// TIA Portal V18 export
ORGANIZATION_BLOCK "Work Cyclic"   // OB30, LAD, CyclicInterrupt
TITLE = Description:
{ S7_Optimized_Access := 'TRUE' }
VERSION : 0.1
// Operations that are supposed to be executed in a precise cycle time, which is temporary set to 45ms. It is important to connect this time with the read/write time of the WebDB (NOAH).
// stored: AutoNumber true, IsIECCheckEnabled false, SetENOAutomatically false
   VAR_INPUT
      Initial_Call : Bool;   // Initial call of this OB
      Event_Count : Int;   // Events discarded
   END_VAR
   VAR_TEMP   // added for the SCL form of the ladder/FBD networks
      _w1 : Bool;
   END_VAR
BEGIN

REGION Network 1: AXIS Z1 Control CMMT V2 To Update
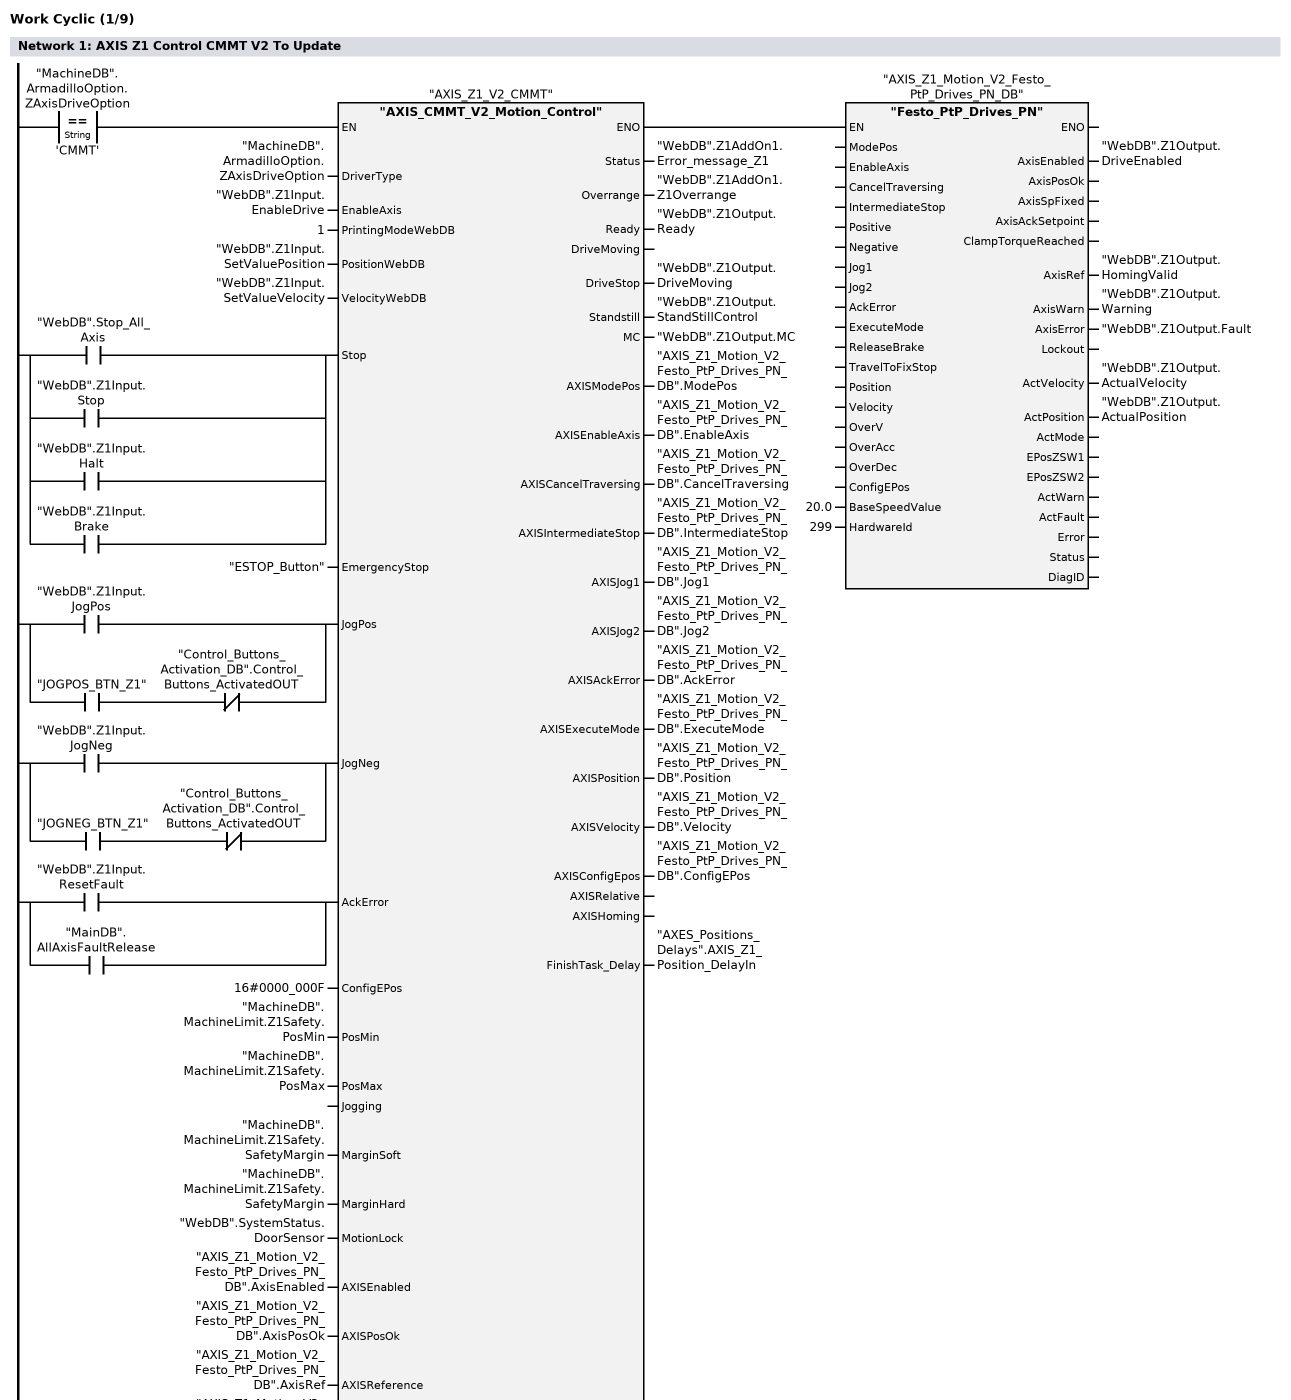
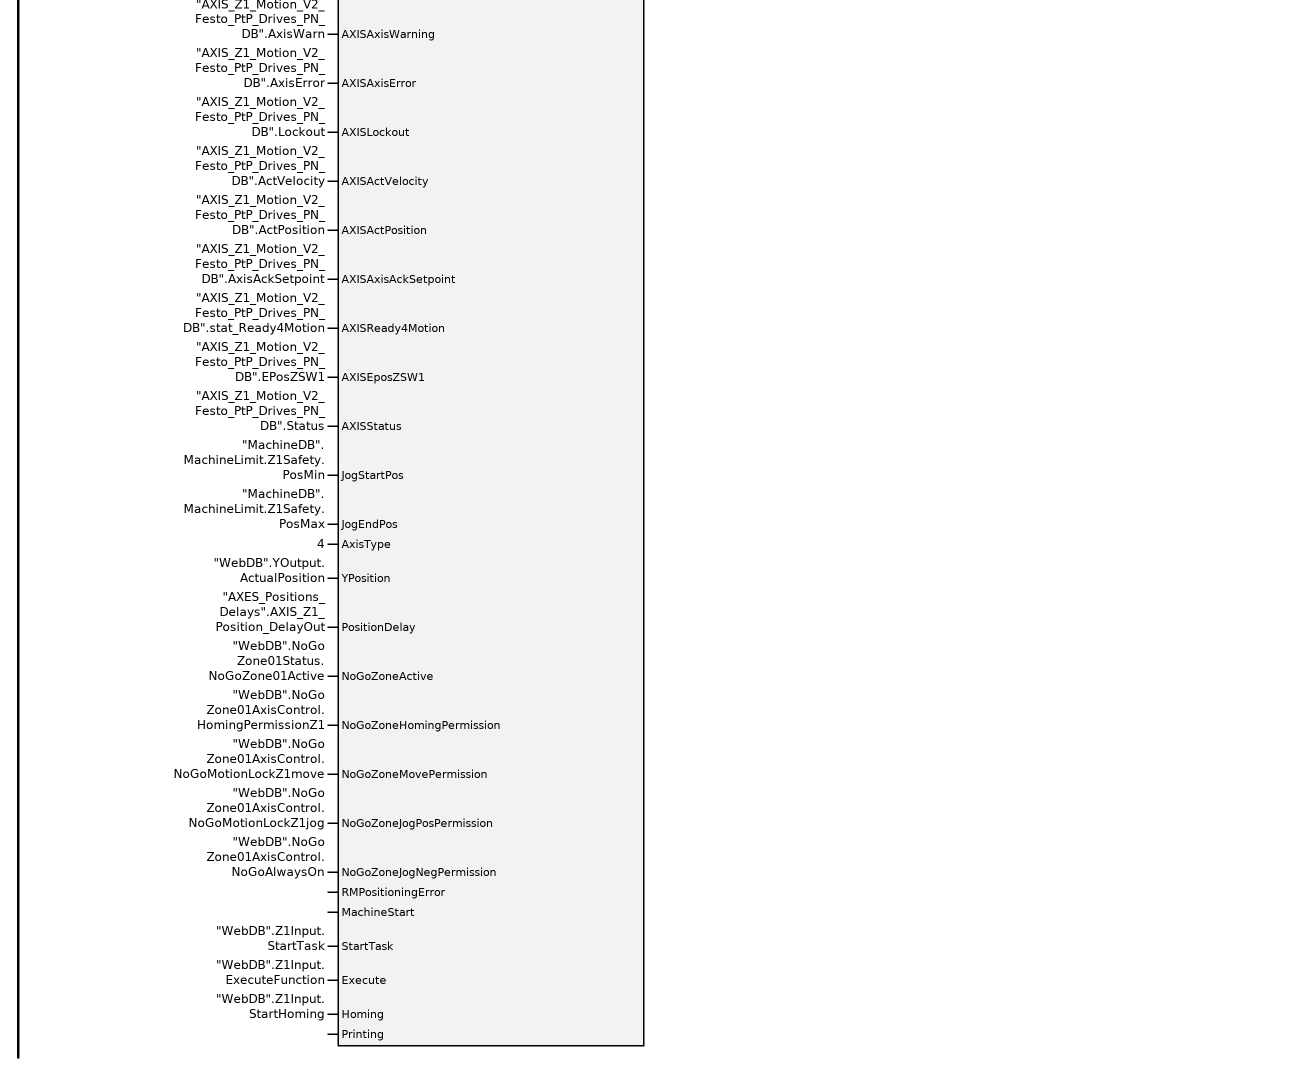
   RUNG wire#powerrail
      { S7_Templates := "SrcType := String" } EQ_Contact(in1 := "MachineDB".ArmadilloOption.ZAxisDriveOption, in2 := 'CMMT')
      "AXIS_Z1_V2_CMMT"(Stop := wire#w1, JogPos := wire#w2, JogNeg := wire#w3, AckError := wire#w4, DriverType := "MachineDB".ArmadilloOption.ZAxisDriveOption, EnableAxis := "WebDB".Z1Input.EnableDrive, PrintingModeWebDB := 1, PositionWebDB := "WebDB".Z1Input.SetValuePosition, VelocityWebDB := "WebDB".Z1Input.SetValueVelocity, EmergencyStop := "ESTOP_Button", ConfigEPos := 16#0000_000F, PosMin := "MachineDB".MachineLimit.Z1Safety.PosMin, PosMax := "MachineDB".MachineLimit.Z1Safety.PosMax, Jogging :=, MarginSoft := "MachineDB".MachineLimit.Z1Safety.SafetyMargin, MarginHard := "MachineDB".MachineLimit.Z1Safety.SafetyMargin, MotionLock := "WebDB".SystemStatus.DoorSensor, AXISEnabled := "AXIS_Z1_Motion_V2_Festo_PtP_Drives_PN_DB".AxisEnabled, AXISPosOk := "AXIS_Z1_Motion_V2_Festo_PtP_Drives_PN_DB".AxisPosOk, AXISReference := "AXIS_Z1_Motion_V2_Festo_PtP_Drives_PN_DB".AxisRef, AXISAxisWarning := "AXIS_Z1_Motion_V2_Festo_PtP_Drives_PN_DB".AxisWarn, AXISAxisError := "AXIS_Z1_Motion_V2_Festo_PtP_Drives_PN_DB".AxisError, AXISLockout := "AXIS_Z1_Motion_V2_Festo_PtP_Drives_PN_DB".Lockout, AXISActVelocity := "AXIS_Z1_Motion_V2_Festo_PtP_Drives_PN_DB".ActVelocity, AXISActPosition := "AXIS_Z1_Motion_V2_Festo_PtP_Drives_PN_DB".ActPosition, AXISAxisAckSetpoint := "AXIS_Z1_Motion_V2_Festo_PtP_Drives_PN_DB".AxisAckSetpoint, AXISReady4Motion := "AXIS_Z1_Motion_V2_Festo_PtP_Drives_PN_DB".stat_Ready4Motion, AXISEposZSW1 := "AXIS_Z1_Motion_V2_Festo_PtP_Drives_PN_DB".EPosZSW1, AXISStatus := "AXIS_Z1_Motion_V2_Festo_PtP_Drives_PN_DB".Status, JogStartPos := "MachineDB".MachineLimit.Z1Safety.PosMin, JogEndPos := "MachineDB".MachineLimit.Z1Safety.PosMax, AxisType := 4, YPosition := "WebDB".YOutput.ActualPosition, PositionDelay := "AXES_Positions_Delays".AXIS_Z1_Position_DelayOut, NoGoZoneActive := "WebDB".NoGoZone01Status.NoGoZone01Active, NoGoZoneHomingPermission := "WebDB".NoGoZone01AxisControl.HomingPermissionZ1, NoGoZoneMovePermission := "WebDB".NoGoZone01AxisControl.NoGoMotionLockZ1move, NoGoZoneJogPosPermission := "WebDB".NoGoZone01AxisControl.NoGoMotionLockZ1jog, NoGoZoneJogNegPermission := "WebDB".NoGoZone01AxisControl.NoGoAlwaysOn, RMPositioningError :=, MachineStart :=, StartTask := "WebDB".Z1Input.StartTask, Execute := "WebDB".Z1Input.ExecuteFunction, Homing := "WebDB".Z1Input.StartHoming, Printing :=, Status => "WebDB".Z1AddOn1.Error_message_Z1, Overrange => "WebDB".Z1AddOn1.Z1Overrange, Ready => "WebDB".Z1Output.Ready, DriveMoving =>, DriveStop => "WebDB".Z1Output.DriveMoving, Standstill => "WebDB".Z1Output.StandStillControl, MC => "WebDB".Z1Output.MC, AXISModePos => "AXIS_Z1_Motion_V2_Festo_PtP_Drives_PN_DB".ModePos, AXISEnableAxis => "AXIS_Z1_Motion_V2_Festo_PtP_Drives_PN_DB".EnableAxis, AXISCancelTraversing => "AXIS_Z1_Motion_V2_Festo_PtP_Drives_PN_DB".CancelTraversing, AXISIntermediateStop => "AXIS_Z1_Motion_V2_Festo_PtP_Drives_PN_DB".IntermediateStop, AXISJog1 => "AXIS_Z1_Motion_V2_Festo_PtP_Drives_PN_DB".Jog1, AXISJog2 => "AXIS_Z1_Motion_V2_Festo_PtP_Drives_PN_DB".Jog2, AXISAckError => "AXIS_Z1_Motion_V2_Festo_PtP_Drives_PN_DB".AckError, AXISExecuteMode => "AXIS_Z1_Motion_V2_Festo_PtP_Drives_PN_DB".ExecuteMode, AXISPosition => "AXIS_Z1_Motion_V2_Festo_PtP_Drives_PN_DB".Position, AXISVelocity => "AXIS_Z1_Motion_V2_Festo_PtP_Drives_PN_DB".Velocity, AXISConfigEpos => "AXIS_Z1_Motion_V2_Festo_PtP_Drives_PN_DB".ConfigEPos, AXISRelative =>, AXISHoming =>, FinishTask_Delay => "AXES_Positions_Delays".AXIS_Z1_Position_DelayIn)
      "AXIS_Z1_Motion_V2_Festo_PtP_Drives_PN_DB"(ModePos :=, EnableAxis :=, CancelTraversing :=, IntermediateStop :=, Positive :=, Negative :=, Jog1 :=, Jog2 :=, AckError :=, ExecuteMode :=, ReleaseBrake :=, TravelToFixStop :=, Position :=, Velocity :=, OverV :=, OverAcc :=, OverDec :=, ConfigEPos :=, BaseSpeedValue := 20.0, HardwareId := 299, AxisEnabled => "WebDB".Z1Output.DriveEnabled, AxisPosOk =>, AxisSpFixed =>, AxisAckSetpoint =>, ClampTorqueReached =>, AxisRef => "WebDB".Z1Output.HomingValid, AxisWarn => "WebDB".Z1Output.Warning, AxisError => "WebDB".Z1Output.Fault, Lockout =>, ActVelocity => "WebDB".Z1Output.ActualVelocity, ActPosition => "WebDB".Z1Output.ActualPosition, ActMode =>, EPosZSW1 =>, EPosZSW2 =>, ActWarn =>, ActFault =>, Error =>, Status =>, DiagID =>)
   END_RUNG
   RUNG wire#powerrail
      Contact( "WebDB".Stop_All_Axis )
   END_RUNG wire#w1
   RUNG wire#powerrail
      Contact( "WebDB".Z1Input.Stop )
   END_RUNG wire#w1
   RUNG wire#powerrail
      Contact( "WebDB".Z1Input.Halt )
   END_RUNG wire#w1
   RUNG wire#powerrail
      Contact( "WebDB".Z1Input.Brake )
   END_RUNG wire#w1
   RUNG wire#powerrail
      Contact( "WebDB".Z1Input.JogPos )
   END_RUNG wire#w2
   RUNG wire#powerrail
      Contact( "JOGPOS_BTN_Z1" )
      I_Contact( "Control_Buttons_Activation_DB".Control_Buttons_ActivatedOUT )
   END_RUNG wire#w2
   RUNG wire#powerrail
      Contact( "WebDB".Z1Input.JogNeg )
   END_RUNG wire#w3
   RUNG wire#powerrail
      Contact( "JOGNEG_BTN_Z1" )
      I_Contact( "Control_Buttons_Activation_DB".Control_Buttons_ActivatedOUT )
   END_RUNG wire#w3
   RUNG wire#powerrail
      Contact( "WebDB".Z1Input.ResetFault )
   END_RUNG wire#w4
   RUNG wire#powerrail
      Contact( "MainDB".AllAxisFaultRelease )
   END_RUNG wire#w4
   // the same network as SCL:
   "AXIS_Z1_V2_CMMT"(EN := "MachineDB".ArmadilloOption.ZAxisDriveOption = 'CMMT',   // "AXIS_CMMT_V2_Motion_Control"
                     DriverType := "MachineDB".ArmadilloOption.ZAxisDriveOption,
                     EnableAxis := "WebDB".Z1Input.EnableDrive,
                     PrintingModeWebDB := 1,
                     PositionWebDB := "WebDB".Z1Input.SetValuePosition,
                     VelocityWebDB := "WebDB".Z1Input.SetValueVelocity,
                     Stop := "WebDB".Stop_All_Axis OR "WebDB".Z1Input.Stop OR "WebDB".Z1Input.Halt OR "WebDB".Z1Input.Brake,
                     EmergencyStop := "ESTOP_Button",
                     JogPos := "WebDB".Z1Input.JogPos OR ("JOGPOS_BTN_Z1" AND NOT "Control_Buttons_Activation_DB".Control_Buttons_ActivatedOUT),
                     JogNeg := "WebDB".Z1Input.JogNeg OR ("JOGNEG_BTN_Z1" AND NOT "Control_Buttons_Activation_DB".Control_Buttons_ActivatedOUT),
                     AckError := "WebDB".Z1Input.ResetFault OR "MainDB".AllAxisFaultRelease,
                     ConfigEPos := 16#0000_000F,
                     PosMin := "MachineDB".MachineLimit.Z1Safety.PosMin,
                     PosMax := "MachineDB".MachineLimit.Z1Safety.PosMax,
                     MarginSoft := "MachineDB".MachineLimit.Z1Safety.SafetyMargin,
                     MarginHard := "MachineDB".MachineLimit.Z1Safety.SafetyMargin,
                     MotionLock := "WebDB".SystemStatus.DoorSensor,
                     AXISEnabled := "AXIS_Z1_Motion_V2_Festo_PtP_Drives_PN_DB".AxisEnabled,
                     AXISPosOk := "AXIS_Z1_Motion_V2_Festo_PtP_Drives_PN_DB".AxisPosOk,
                     AXISReference := "AXIS_Z1_Motion_V2_Festo_PtP_Drives_PN_DB".AxisRef,
                     AXISAxisWarning := "AXIS_Z1_Motion_V2_Festo_PtP_Drives_PN_DB".AxisWarn,
                     AXISAxisError := "AXIS_Z1_Motion_V2_Festo_PtP_Drives_PN_DB".AxisError,
                     AXISLockout := "AXIS_Z1_Motion_V2_Festo_PtP_Drives_PN_DB".Lockout,
                     AXISActVelocity := "AXIS_Z1_Motion_V2_Festo_PtP_Drives_PN_DB".ActVelocity,
                     AXISActPosition := "AXIS_Z1_Motion_V2_Festo_PtP_Drives_PN_DB".ActPosition,
                     AXISAxisAckSetpoint := "AXIS_Z1_Motion_V2_Festo_PtP_Drives_PN_DB".AxisAckSetpoint,
                     AXISReady4Motion := "AXIS_Z1_Motion_V2_Festo_PtP_Drives_PN_DB".stat_Ready4Motion,
                     AXISEposZSW1 := "AXIS_Z1_Motion_V2_Festo_PtP_Drives_PN_DB".EPosZSW1,
                     AXISStatus := "AXIS_Z1_Motion_V2_Festo_PtP_Drives_PN_DB".Status,
                     JogStartPos := "MachineDB".MachineLimit.Z1Safety.PosMin,
                     JogEndPos := "MachineDB".MachineLimit.Z1Safety.PosMax,
                     AxisType := 4,
                     YPosition := "WebDB".YOutput.ActualPosition,
                     PositionDelay := "AXES_Positions_Delays".AXIS_Z1_Position_DelayOut,
                     NoGoZoneActive := "WebDB".NoGoZone01Status.NoGoZone01Active,
                     NoGoZoneHomingPermission := "WebDB".NoGoZone01AxisControl.HomingPermissionZ1,
                     NoGoZoneMovePermission := "WebDB".NoGoZone01AxisControl.NoGoMotionLockZ1move,
                     NoGoZoneJogPosPermission := "WebDB".NoGoZone01AxisControl.NoGoMotionLockZ1jog,
                     NoGoZoneJogNegPermission := "WebDB".NoGoZone01AxisControl.NoGoAlwaysOn,
                     StartTask := "WebDB".Z1Input.StartTask,
                     Execute := "WebDB".Z1Input.ExecuteFunction,
                     Homing := "WebDB".Z1Input.StartHoming,
                     Status => "WebDB".Z1AddOn1.Error_message_Z1,
                     Overrange => "WebDB".Z1AddOn1.Z1Overrange,
                     Ready => "WebDB".Z1Output.Ready,
                     DriveStop => "WebDB".Z1Output.DriveMoving,
                     Standstill => "WebDB".Z1Output.StandStillControl,
                     MC => "WebDB".Z1Output.MC,
                     AXISModePos => "AXIS_Z1_Motion_V2_Festo_PtP_Drives_PN_DB".ModePos,
                     AXISEnableAxis => "AXIS_Z1_Motion_V2_Festo_PtP_Drives_PN_DB".EnableAxis,
                     AXISCancelTraversing => "AXIS_Z1_Motion_V2_Festo_PtP_Drives_PN_DB".CancelTraversing,
                     AXISIntermediateStop => "AXIS_Z1_Motion_V2_Festo_PtP_Drives_PN_DB".IntermediateStop,
                     AXISJog1 => "AXIS_Z1_Motion_V2_Festo_PtP_Drives_PN_DB".Jog1,
                     AXISJog2 => "AXIS_Z1_Motion_V2_Festo_PtP_Drives_PN_DB".Jog2,
                     AXISAckError => "AXIS_Z1_Motion_V2_Festo_PtP_Drives_PN_DB".AckError,
                     AXISExecuteMode => "AXIS_Z1_Motion_V2_Festo_PtP_Drives_PN_DB".ExecuteMode,
                     AXISPosition => "AXIS_Z1_Motion_V2_Festo_PtP_Drives_PN_DB".Position,
                     AXISVelocity => "AXIS_Z1_Motion_V2_Festo_PtP_Drives_PN_DB".Velocity,
                     AXISConfigEpos => "AXIS_Z1_Motion_V2_Festo_PtP_Drives_PN_DB".ConfigEPos,
                     FinishTask_Delay => "AXES_Positions_Delays".AXIS_Z1_Position_DelayIn,
                     ENO => #_w1);
   IF #_w1 THEN
       "AXIS_Z1_Motion_V2_Festo_PtP_Drives_PN_DB"(BaseSpeedValue := 20.0,   // "Festo_PtP_Drives_PN"
                               HardwareId := 299,
                               AxisEnabled => "WebDB".Z1Output.DriveEnabled,
                               AxisRef => "WebDB".Z1Output.HomingValid,
                               AxisWarn => "WebDB".Z1Output.Warning,
                               AxisError => "WebDB".Z1Output.Fault,
                               ActVelocity => "WebDB".Z1Output.ActualVelocity,
                               ActPosition => "WebDB".Z1Output.ActualPosition);
   END_IF;
END_REGION

REGION Network 2: AXIS Z1 Control CMMS
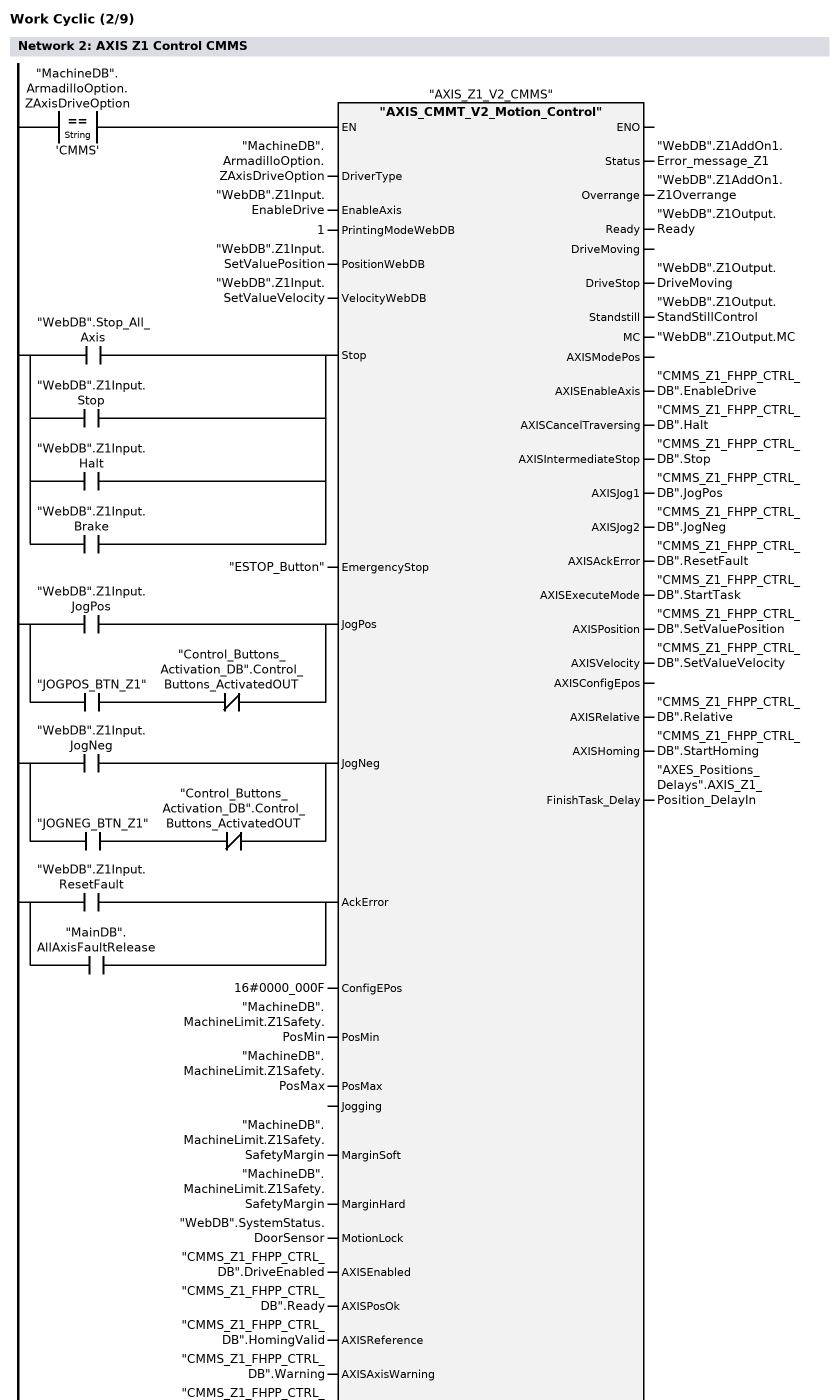
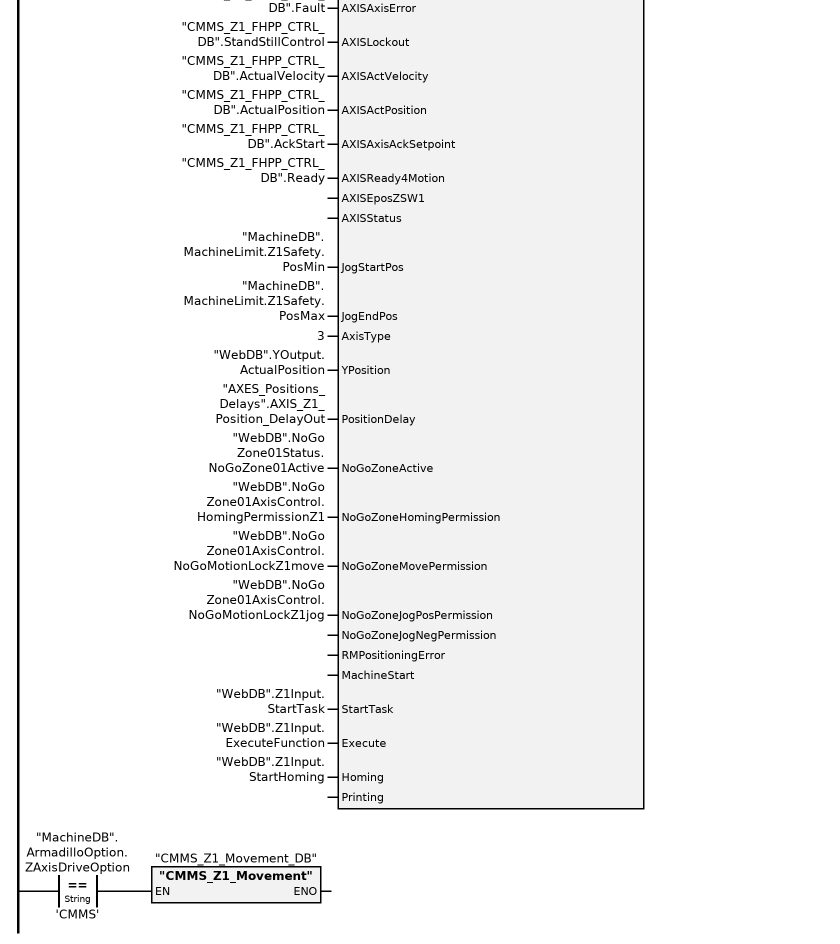
   RUNG wire#powerrail
      { S7_Templates := "SrcType := String" } EQ_Contact(in1 := "MachineDB".ArmadilloOption.ZAxisDriveOption, in2 := 'CMMS')
      "AXIS_Z1_V2_CMMS"(Stop := wire#w1, JogPos := wire#w2, JogNeg := wire#w3, AckError := wire#w4, DriverType := "MachineDB".ArmadilloOption.ZAxisDriveOption, EnableAxis := "WebDB".Z1Input.EnableDrive, PrintingModeWebDB := 1, PositionWebDB := "WebDB".Z1Input.SetValuePosition, VelocityWebDB := "WebDB".Z1Input.SetValueVelocity, EmergencyStop := "ESTOP_Button", ConfigEPos := 16#0000_000F, PosMin := "MachineDB".MachineLimit.Z1Safety.PosMin, PosMax := "MachineDB".MachineLimit.Z1Safety.PosMax, Jogging :=, MarginSoft := "MachineDB".MachineLimit.Z1Safety.SafetyMargin, MarginHard := "MachineDB".MachineLimit.Z1Safety.SafetyMargin, MotionLock := "WebDB".SystemStatus.DoorSensor, AXISEnabled := "CMMS_Z1_FHPP_CTRL_DB".DriveEnabled, AXISPosOk := "CMMS_Z1_FHPP_CTRL_DB".Ready, AXISReference := "CMMS_Z1_FHPP_CTRL_DB".HomingValid, AXISAxisWarning := "CMMS_Z1_FHPP_CTRL_DB".Warning, AXISAxisError := "CMMS_Z1_FHPP_CTRL_DB".Fault, AXISLockout := "CMMS_Z1_FHPP_CTRL_DB".StandStillControl, AXISActVelocity := "CMMS_Z1_FHPP_CTRL_DB".ActualVelocity, AXISActPosition := "CMMS_Z1_FHPP_CTRL_DB".ActualPosition, AXISAxisAckSetpoint := "CMMS_Z1_FHPP_CTRL_DB".AckStart, AXISReady4Motion := "CMMS_Z1_FHPP_CTRL_DB".Ready, AXISEposZSW1 :=, AXISStatus :=, JogStartPos := "MachineDB".MachineLimit.Z1Safety.PosMin, JogEndPos := "MachineDB".MachineLimit.Z1Safety.PosMax, AxisType := 3, YPosition := "WebDB".YOutput.ActualPosition, PositionDelay := "AXES_Positions_Delays".AXIS_Z1_Position_DelayOut, NoGoZoneActive := "WebDB".NoGoZone01Status.NoGoZone01Active, NoGoZoneHomingPermission := "WebDB".NoGoZone01AxisControl.HomingPermissionZ1, NoGoZoneMovePermission := "WebDB".NoGoZone01AxisControl.NoGoMotionLockZ1move, NoGoZoneJogPosPermission := "WebDB".NoGoZone01AxisControl.NoGoMotionLockZ1jog, NoGoZoneJogNegPermission :=, RMPositioningError :=, MachineStart :=, StartTask := "WebDB".Z1Input.StartTask, Execute := "WebDB".Z1Input.ExecuteFunction, Homing := "WebDB".Z1Input.StartHoming, Printing :=, Status => "WebDB".Z1AddOn1.Error_message_Z1, Overrange => "WebDB".Z1AddOn1.Z1Overrange, Ready => "WebDB".Z1Output.Ready, DriveMoving =>, DriveStop => "WebDB".Z1Output.DriveMoving, Standstill => "WebDB".Z1Output.StandStillControl, MC => "WebDB".Z1Output.MC, AXISModePos =>, AXISEnableAxis => "CMMS_Z1_FHPP_CTRL_DB".EnableDrive, AXISCancelTraversing => "CMMS_Z1_FHPP_CTRL_DB".Halt, AXISIntermediateStop => "CMMS_Z1_FHPP_CTRL_DB".Stop, AXISJog1 => "CMMS_Z1_FHPP_CTRL_DB".JogPos, AXISJog2 => "CMMS_Z1_FHPP_CTRL_DB".JogNeg, AXISAckError => "CMMS_Z1_FHPP_CTRL_DB".ResetFault, AXISExecuteMode => "CMMS_Z1_FHPP_CTRL_DB".StartTask, AXISPosition => "CMMS_Z1_FHPP_CTRL_DB".SetValuePosition, AXISVelocity => "CMMS_Z1_FHPP_CTRL_DB".SetValueVelocity, AXISConfigEpos =>, AXISRelative => "CMMS_Z1_FHPP_CTRL_DB".Relative, AXISHoming => "CMMS_Z1_FHPP_CTRL_DB".StartHoming, FinishTask_Delay => "AXES_Positions_Delays".AXIS_Z1_Position_DelayIn)
   END_RUNG
   RUNG wire#powerrail
      Contact( "WebDB".Stop_All_Axis )
   END_RUNG wire#w1
   RUNG wire#powerrail
      Contact( "WebDB".Z1Input.Stop )
   END_RUNG wire#w1
   RUNG wire#powerrail
      Contact( "WebDB".Z1Input.Halt )
   END_RUNG wire#w1
   RUNG wire#powerrail
      Contact( "WebDB".Z1Input.Brake )
   END_RUNG wire#w1
   RUNG wire#powerrail
      Contact( "WebDB".Z1Input.JogPos )
   END_RUNG wire#w2
   RUNG wire#powerrail
      Contact( "JOGPOS_BTN_Z1" )
      I_Contact( "Control_Buttons_Activation_DB".Control_Buttons_ActivatedOUT )
   END_RUNG wire#w2
   RUNG wire#powerrail
      Contact( "WebDB".Z1Input.JogNeg )
   END_RUNG wire#w3
   RUNG wire#powerrail
      Contact( "JOGNEG_BTN_Z1" )
      I_Contact( "Control_Buttons_Activation_DB".Control_Buttons_ActivatedOUT )
   END_RUNG wire#w3
   RUNG wire#powerrail
      Contact( "WebDB".Z1Input.ResetFault )
   END_RUNG wire#w4
   RUNG wire#powerrail
      Contact( "MainDB".AllAxisFaultRelease )
   END_RUNG wire#w4
   RUNG wire#powerrail
      { S7_Templates := "SrcType := String" } EQ_Contact(in1 := "MachineDB".ArmadilloOption.ZAxisDriveOption, in2 := 'CMMS')
      "CMMS_Z1_Movement_DB"()
   END_RUNG
   // the same network as SCL:
   IF "MachineDB".ArmadilloOption.ZAxisDriveOption = 'CMMS' THEN
       "AXIS_Z1_V2_CMMS"(DriverType := "MachineDB".ArmadilloOption.ZAxisDriveOption,   // "AXIS_CMMT_V2_Motion_Control"
                         EnableAxis := "WebDB".Z1Input.EnableDrive,
                         PrintingModeWebDB := 1,
                         PositionWebDB := "WebDB".Z1Input.SetValuePosition,
                         VelocityWebDB := "WebDB".Z1Input.SetValueVelocity,
                         Stop := "WebDB".Stop_All_Axis OR "WebDB".Z1Input.Stop OR "WebDB".Z1Input.Halt OR "WebDB".Z1Input.Brake,
                         EmergencyStop := "ESTOP_Button",
                         JogPos := "WebDB".Z1Input.JogPos OR ("JOGPOS_BTN_Z1" AND NOT "Control_Buttons_Activation_DB".Control_Buttons_ActivatedOUT),
                         JogNeg := "WebDB".Z1Input.JogNeg OR ("JOGNEG_BTN_Z1" AND NOT "Control_Buttons_Activation_DB".Control_Buttons_ActivatedOUT),
                         AckError := "WebDB".Z1Input.ResetFault OR "MainDB".AllAxisFaultRelease,
                         ConfigEPos := 16#0000_000F,
                         PosMin := "MachineDB".MachineLimit.Z1Safety.PosMin,
                         PosMax := "MachineDB".MachineLimit.Z1Safety.PosMax,
                         MarginSoft := "MachineDB".MachineLimit.Z1Safety.SafetyMargin,
                         MarginHard := "MachineDB".MachineLimit.Z1Safety.SafetyMargin,
                         MotionLock := "WebDB".SystemStatus.DoorSensor,
                         AXISEnabled := "CMMS_Z1_FHPP_CTRL_DB".DriveEnabled,
                         AXISPosOk := "CMMS_Z1_FHPP_CTRL_DB".Ready,
                         AXISReference := "CMMS_Z1_FHPP_CTRL_DB".HomingValid,
                         AXISAxisWarning := "CMMS_Z1_FHPP_CTRL_DB".Warning,
                         AXISAxisError := "CMMS_Z1_FHPP_CTRL_DB".Fault,
                         AXISLockout := "CMMS_Z1_FHPP_CTRL_DB".StandStillControl,
                         AXISActVelocity := "CMMS_Z1_FHPP_CTRL_DB".ActualVelocity,
                         AXISActPosition := "CMMS_Z1_FHPP_CTRL_DB".ActualPosition,
                         AXISAxisAckSetpoint := "CMMS_Z1_FHPP_CTRL_DB".AckStart,
                         AXISReady4Motion := "CMMS_Z1_FHPP_CTRL_DB".Ready,
                         JogStartPos := "MachineDB".MachineLimit.Z1Safety.PosMin,
                         JogEndPos := "MachineDB".MachineLimit.Z1Safety.PosMax,
                         AxisType := 3,
                         YPosition := "WebDB".YOutput.ActualPosition,
                         PositionDelay := "AXES_Positions_Delays".AXIS_Z1_Position_DelayOut,
                         NoGoZoneActive := "WebDB".NoGoZone01Status.NoGoZone01Active,
                         NoGoZoneHomingPermission := "WebDB".NoGoZone01AxisControl.HomingPermissionZ1,
                         NoGoZoneMovePermission := "WebDB".NoGoZone01AxisControl.NoGoMotionLockZ1move,
                         NoGoZoneJogPosPermission := "WebDB".NoGoZone01AxisControl.NoGoMotionLockZ1jog,
                         StartTask := "WebDB".Z1Input.StartTask,
                         Execute := "WebDB".Z1Input.ExecuteFunction,
                         Homing := "WebDB".Z1Input.StartHoming,
                         Status => "WebDB".Z1AddOn1.Error_message_Z1,
                         Overrange => "WebDB".Z1AddOn1.Z1Overrange,
                         Ready => "WebDB".Z1Output.Ready,
                         DriveStop => "WebDB".Z1Output.DriveMoving,
                         Standstill => "WebDB".Z1Output.StandStillControl,
                         MC => "WebDB".Z1Output.MC,
                         AXISEnableAxis => "CMMS_Z1_FHPP_CTRL_DB".EnableDrive,
                         AXISCancelTraversing => "CMMS_Z1_FHPP_CTRL_DB".Halt,
                         AXISIntermediateStop => "CMMS_Z1_FHPP_CTRL_DB".Stop,
                         AXISJog1 => "CMMS_Z1_FHPP_CTRL_DB".JogPos,
                         AXISJog2 => "CMMS_Z1_FHPP_CTRL_DB".JogNeg,
                         AXISAckError => "CMMS_Z1_FHPP_CTRL_DB".ResetFault,
                         AXISExecuteMode => "CMMS_Z1_FHPP_CTRL_DB".StartTask,
                         AXISPosition => "CMMS_Z1_FHPP_CTRL_DB".SetValuePosition,
                         AXISVelocity => "CMMS_Z1_FHPP_CTRL_DB".SetValueVelocity,
                         AXISRelative => "CMMS_Z1_FHPP_CTRL_DB".Relative,
                         AXISHoming => "CMMS_Z1_FHPP_CTRL_DB".StartHoming,
                         FinishTask_Delay => "AXES_Positions_Delays".AXIS_Z1_Position_DelayIn);
   END_IF;
   IF "MachineDB".ArmadilloOption.ZAxisDriveOption = 'CMMS' THEN
       "CMMS_Z1_Movement_DB"();   // "CMMS_Z1_Movement"
   END_IF;
END_REGION

REGION Network 3: AXIZ Z1 Delays
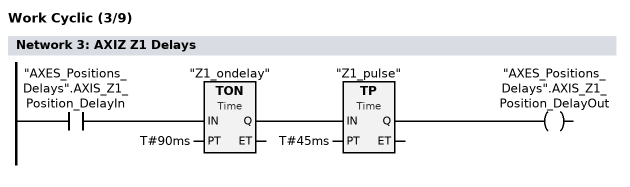
   RUNG wire#powerrail
      Contact( "AXES_Positions_Delays".AXIS_Z1_Position_DelayIn )
      { S7_Templates := "time_type := Time" } "Z1_ondelay".TON(pt := T#90ms, et =>)
      { S7_Templates := "time_type := Time" } "Z1_pulse".TP(pt := T#45ms, et =>)
      Coil( "AXES_Positions_Delays".AXIS_Z1_Position_DelayOut )
   END_RUNG
   // the same network as SCL:
   "Z1_ondelay".TON(IN := "AXES_Positions_Delays".AXIS_Z1_Position_DelayIn, PT := T#90ms);
   "Z1_pulse".TP(IN := "Z1_ondelay".Q, PT := T#45ms);
   "AXES_Positions_Delays".AXIS_Z1_Position_DelayOut := "Z1_pulse".Q;
END_REGION

REGION Network 4: AXIS Z2 Control CMMT V2 To Update
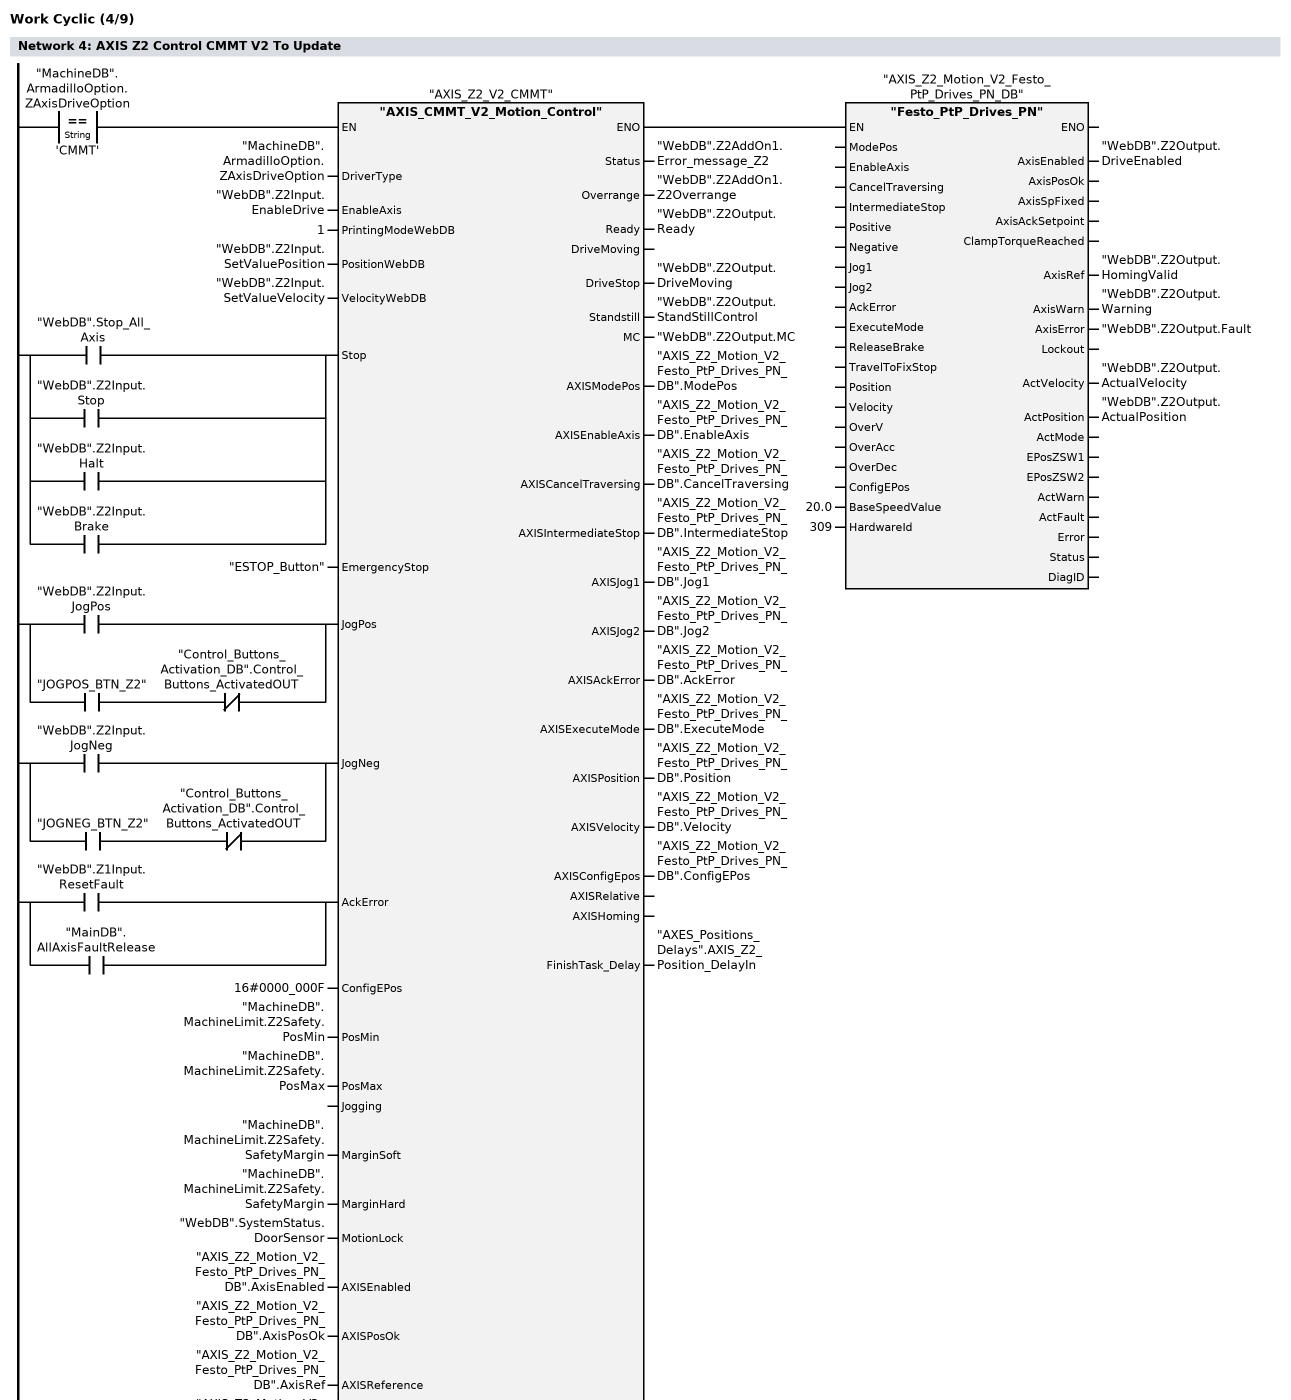
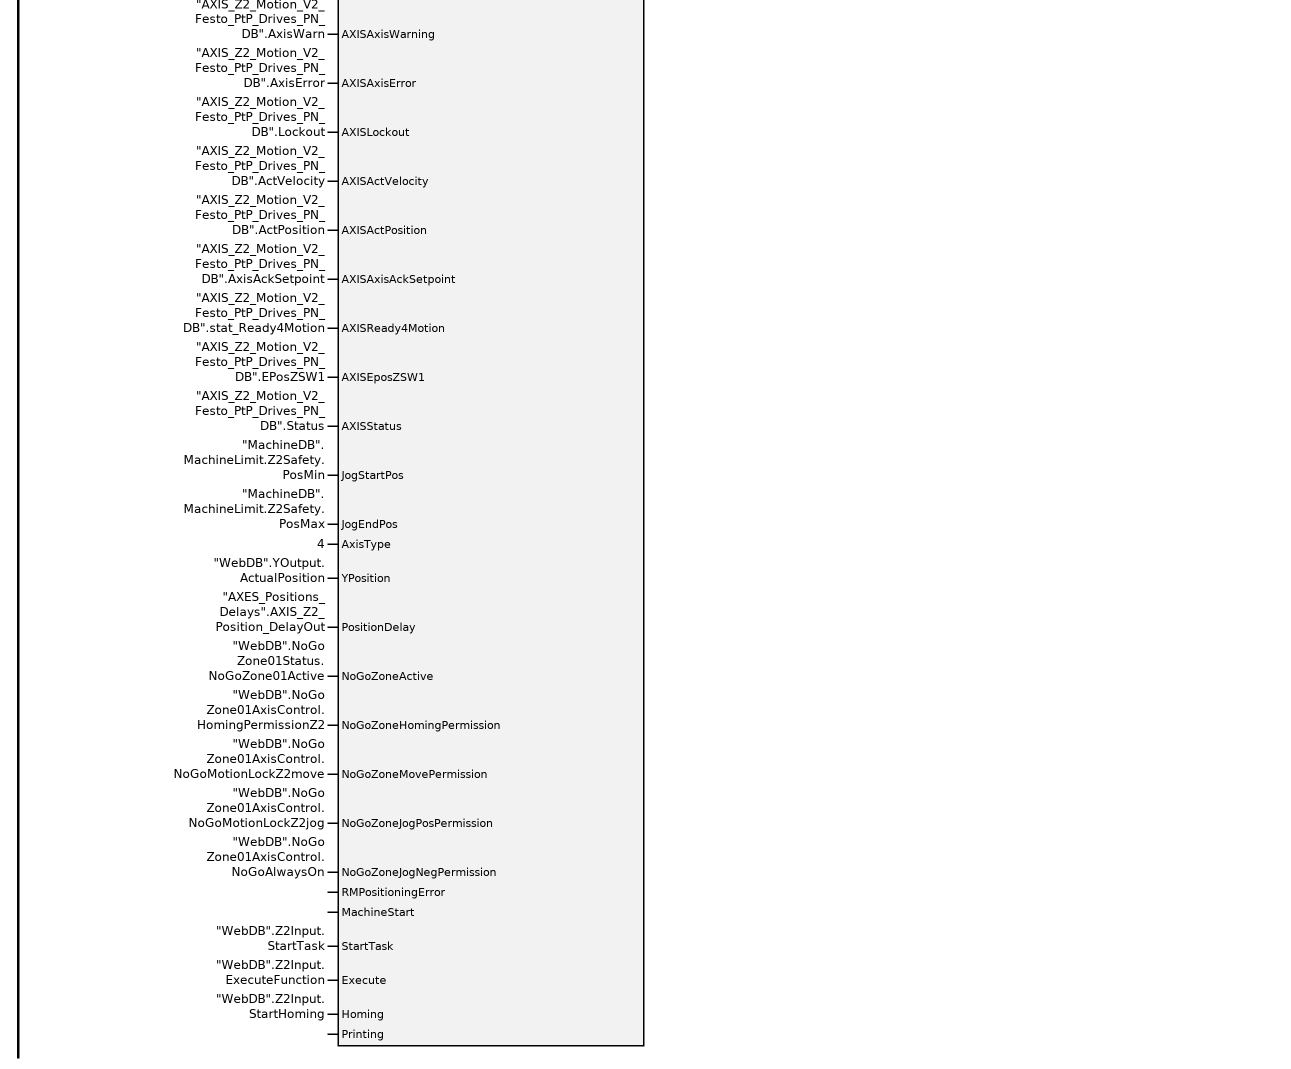
   RUNG wire#powerrail
      { S7_Templates := "SrcType := String" } EQ_Contact(in1 := "MachineDB".ArmadilloOption.ZAxisDriveOption, in2 := 'CMMT')
      "AXIS_Z2_V2_CMMT"(Stop := wire#w1, JogPos := wire#w2, JogNeg := wire#w3, AckError := wire#w4, DriverType := "MachineDB".ArmadilloOption.ZAxisDriveOption, EnableAxis := "WebDB".Z2Input.EnableDrive, PrintingModeWebDB := 1, PositionWebDB := "WebDB".Z2Input.SetValuePosition, VelocityWebDB := "WebDB".Z2Input.SetValueVelocity, EmergencyStop := "ESTOP_Button", ConfigEPos := 16#0000_000F, PosMin := "MachineDB".MachineLimit.Z2Safety.PosMin, PosMax := "MachineDB".MachineLimit.Z2Safety.PosMax, Jogging :=, MarginSoft := "MachineDB".MachineLimit.Z2Safety.SafetyMargin, MarginHard := "MachineDB".MachineLimit.Z2Safety.SafetyMargin, MotionLock := "WebDB".SystemStatus.DoorSensor, AXISEnabled := "AXIS_Z2_Motion_V2_Festo_PtP_Drives_PN_DB".AxisEnabled, AXISPosOk := "AXIS_Z2_Motion_V2_Festo_PtP_Drives_PN_DB".AxisPosOk, AXISReference := "AXIS_Z2_Motion_V2_Festo_PtP_Drives_PN_DB".AxisRef, AXISAxisWarning := "AXIS_Z2_Motion_V2_Festo_PtP_Drives_PN_DB".AxisWarn, AXISAxisError := "AXIS_Z2_Motion_V2_Festo_PtP_Drives_PN_DB".AxisError, AXISLockout := "AXIS_Z2_Motion_V2_Festo_PtP_Drives_PN_DB".Lockout, AXISActVelocity := "AXIS_Z2_Motion_V2_Festo_PtP_Drives_PN_DB".ActVelocity, AXISActPosition := "AXIS_Z2_Motion_V2_Festo_PtP_Drives_PN_DB".ActPosition, AXISAxisAckSetpoint := "AXIS_Z2_Motion_V2_Festo_PtP_Drives_PN_DB".AxisAckSetpoint, AXISReady4Motion := "AXIS_Z2_Motion_V2_Festo_PtP_Drives_PN_DB".stat_Ready4Motion, AXISEposZSW1 := "AXIS_Z2_Motion_V2_Festo_PtP_Drives_PN_DB".EPosZSW1, AXISStatus := "AXIS_Z2_Motion_V2_Festo_PtP_Drives_PN_DB".Status, JogStartPos := "MachineDB".MachineLimit.Z2Safety.PosMin, JogEndPos := "MachineDB".MachineLimit.Z2Safety.PosMax, AxisType := 4, YPosition := "WebDB".YOutput.ActualPosition, PositionDelay := "AXES_Positions_Delays".AXIS_Z2_Position_DelayOut, NoGoZoneActive := "WebDB".NoGoZone01Status.NoGoZone01Active, NoGoZoneHomingPermission := "WebDB".NoGoZone01AxisControl.HomingPermissionZ2, NoGoZoneMovePermission := "WebDB".NoGoZone01AxisControl.NoGoMotionLockZ2move, NoGoZoneJogPosPermission := "WebDB".NoGoZone01AxisControl.NoGoMotionLockZ2jog, NoGoZoneJogNegPermission := "WebDB".NoGoZone01AxisControl.NoGoAlwaysOn, RMPositioningError :=, MachineStart :=, StartTask := "WebDB".Z2Input.StartTask, Execute := "WebDB".Z2Input.ExecuteFunction, Homing := "WebDB".Z2Input.StartHoming, Printing :=, Status => "WebDB".Z2AddOn1.Error_message_Z2, Overrange => "WebDB".Z2AddOn1.Z2Overrange, Ready => "WebDB".Z2Output.Ready, DriveMoving =>, DriveStop => "WebDB".Z2Output.DriveMoving, Standstill => "WebDB".Z2Output.StandStillControl, MC => "WebDB".Z2Output.MC, AXISModePos => "AXIS_Z2_Motion_V2_Festo_PtP_Drives_PN_DB".ModePos, AXISEnableAxis => "AXIS_Z2_Motion_V2_Festo_PtP_Drives_PN_DB".EnableAxis, AXISCancelTraversing => "AXIS_Z2_Motion_V2_Festo_PtP_Drives_PN_DB".CancelTraversing, AXISIntermediateStop => "AXIS_Z2_Motion_V2_Festo_PtP_Drives_PN_DB".IntermediateStop, AXISJog1 => "AXIS_Z2_Motion_V2_Festo_PtP_Drives_PN_DB".Jog1, AXISJog2 => "AXIS_Z2_Motion_V2_Festo_PtP_Drives_PN_DB".Jog2, AXISAckError => "AXIS_Z2_Motion_V2_Festo_PtP_Drives_PN_DB".AckError, AXISExecuteMode => "AXIS_Z2_Motion_V2_Festo_PtP_Drives_PN_DB".ExecuteMode, AXISPosition => "AXIS_Z2_Motion_V2_Festo_PtP_Drives_PN_DB".Position, AXISVelocity => "AXIS_Z2_Motion_V2_Festo_PtP_Drives_PN_DB".Velocity, AXISConfigEpos => "AXIS_Z2_Motion_V2_Festo_PtP_Drives_PN_DB".ConfigEPos, AXISRelative =>, AXISHoming =>, FinishTask_Delay => "AXES_Positions_Delays".AXIS_Z2_Position_DelayIn)
      "AXIS_Z2_Motion_V2_Festo_PtP_Drives_PN_DB"(ModePos :=, EnableAxis :=, CancelTraversing :=, IntermediateStop :=, Positive :=, Negative :=, Jog1 :=, Jog2 :=, AckError :=, ExecuteMode :=, ReleaseBrake :=, TravelToFixStop :=, Position :=, Velocity :=, OverV :=, OverAcc :=, OverDec :=, ConfigEPos :=, BaseSpeedValue := 20.0, HardwareId := 309, AxisEnabled => "WebDB".Z2Output.DriveEnabled, AxisPosOk =>, AxisSpFixed =>, AxisAckSetpoint =>, ClampTorqueReached =>, AxisRef => "WebDB".Z2Output.HomingValid, AxisWarn => "WebDB".Z2Output.Warning, AxisError => "WebDB".Z2Output.Fault, Lockout =>, ActVelocity => "WebDB".Z2Output.ActualVelocity, ActPosition => "WebDB".Z2Output.ActualPosition, ActMode =>, EPosZSW1 =>, EPosZSW2 =>, ActWarn =>, ActFault =>, Error =>, Status =>, DiagID =>)
   END_RUNG
   RUNG wire#powerrail
      Contact( "WebDB".Stop_All_Axis )
   END_RUNG wire#w1
   RUNG wire#powerrail
      Contact( "WebDB".Z2Input.Stop )
   END_RUNG wire#w1
   RUNG wire#powerrail
      Contact( "WebDB".Z2Input.Halt )
   END_RUNG wire#w1
   RUNG wire#powerrail
      Contact( "WebDB".Z2Input.Brake )
   END_RUNG wire#w1
   RUNG wire#powerrail
      Contact( "WebDB".Z2Input.JogPos )
   END_RUNG wire#w2
   RUNG wire#powerrail
      Contact( "JOGPOS_BTN_Z2" )
      I_Contact( "Control_Buttons_Activation_DB".Control_Buttons_ActivatedOUT )
   END_RUNG wire#w2
   RUNG wire#powerrail
      Contact( "WebDB".Z2Input.JogNeg )
   END_RUNG wire#w3
   RUNG wire#powerrail
      Contact( "JOGNEG_BTN_Z2" )
      I_Contact( "Control_Buttons_Activation_DB".Control_Buttons_ActivatedOUT )
   END_RUNG wire#w3
   RUNG wire#powerrail
      Contact( "WebDB".Z1Input.ResetFault )
   END_RUNG wire#w4
   RUNG wire#powerrail
      Contact( "MainDB".AllAxisFaultRelease )
   END_RUNG wire#w4
   // the same network as SCL:
   "AXIS_Z2_V2_CMMT"(EN := "MachineDB".ArmadilloOption.ZAxisDriveOption = 'CMMT',   // "AXIS_CMMT_V2_Motion_Control"
                     DriverType := "MachineDB".ArmadilloOption.ZAxisDriveOption,
                     EnableAxis := "WebDB".Z2Input.EnableDrive,
                     PrintingModeWebDB := 1,
                     PositionWebDB := "WebDB".Z2Input.SetValuePosition,
                     VelocityWebDB := "WebDB".Z2Input.SetValueVelocity,
                     Stop := "WebDB".Stop_All_Axis OR "WebDB".Z2Input.Stop OR "WebDB".Z2Input.Halt OR "WebDB".Z2Input.Brake,
                     EmergencyStop := "ESTOP_Button",
                     JogPos := "WebDB".Z2Input.JogPos OR ("JOGPOS_BTN_Z2" AND NOT "Control_Buttons_Activation_DB".Control_Buttons_ActivatedOUT),
                     JogNeg := "WebDB".Z2Input.JogNeg OR ("JOGNEG_BTN_Z2" AND NOT "Control_Buttons_Activation_DB".Control_Buttons_ActivatedOUT),
                     AckError := "WebDB".Z1Input.ResetFault OR "MainDB".AllAxisFaultRelease,
                     ConfigEPos := 16#0000_000F,
                     PosMin := "MachineDB".MachineLimit.Z2Safety.PosMin,
                     PosMax := "MachineDB".MachineLimit.Z2Safety.PosMax,
                     MarginSoft := "MachineDB".MachineLimit.Z2Safety.SafetyMargin,
                     MarginHard := "MachineDB".MachineLimit.Z2Safety.SafetyMargin,
                     MotionLock := "WebDB".SystemStatus.DoorSensor,
                     AXISEnabled := "AXIS_Z2_Motion_V2_Festo_PtP_Drives_PN_DB".AxisEnabled,
                     AXISPosOk := "AXIS_Z2_Motion_V2_Festo_PtP_Drives_PN_DB".AxisPosOk,
                     AXISReference := "AXIS_Z2_Motion_V2_Festo_PtP_Drives_PN_DB".AxisRef,
                     AXISAxisWarning := "AXIS_Z2_Motion_V2_Festo_PtP_Drives_PN_DB".AxisWarn,
                     AXISAxisError := "AXIS_Z2_Motion_V2_Festo_PtP_Drives_PN_DB".AxisError,
                     AXISLockout := "AXIS_Z2_Motion_V2_Festo_PtP_Drives_PN_DB".Lockout,
                     AXISActVelocity := "AXIS_Z2_Motion_V2_Festo_PtP_Drives_PN_DB".ActVelocity,
                     AXISActPosition := "AXIS_Z2_Motion_V2_Festo_PtP_Drives_PN_DB".ActPosition,
                     AXISAxisAckSetpoint := "AXIS_Z2_Motion_V2_Festo_PtP_Drives_PN_DB".AxisAckSetpoint,
                     AXISReady4Motion := "AXIS_Z2_Motion_V2_Festo_PtP_Drives_PN_DB".stat_Ready4Motion,
                     AXISEposZSW1 := "AXIS_Z2_Motion_V2_Festo_PtP_Drives_PN_DB".EPosZSW1,
                     AXISStatus := "AXIS_Z2_Motion_V2_Festo_PtP_Drives_PN_DB".Status,
                     JogStartPos := "MachineDB".MachineLimit.Z2Safety.PosMin,
                     JogEndPos := "MachineDB".MachineLimit.Z2Safety.PosMax,
                     AxisType := 4,
                     YPosition := "WebDB".YOutput.ActualPosition,
                     PositionDelay := "AXES_Positions_Delays".AXIS_Z2_Position_DelayOut,
                     NoGoZoneActive := "WebDB".NoGoZone01Status.NoGoZone01Active,
                     NoGoZoneHomingPermission := "WebDB".NoGoZone01AxisControl.HomingPermissionZ2,
                     NoGoZoneMovePermission := "WebDB".NoGoZone01AxisControl.NoGoMotionLockZ2move,
                     NoGoZoneJogPosPermission := "WebDB".NoGoZone01AxisControl.NoGoMotionLockZ2jog,
                     NoGoZoneJogNegPermission := "WebDB".NoGoZone01AxisControl.NoGoAlwaysOn,
                     StartTask := "WebDB".Z2Input.StartTask,
                     Execute := "WebDB".Z2Input.ExecuteFunction,
                     Homing := "WebDB".Z2Input.StartHoming,
                     Status => "WebDB".Z2AddOn1.Error_message_Z2,
                     Overrange => "WebDB".Z2AddOn1.Z2Overrange,
                     Ready => "WebDB".Z2Output.Ready,
                     DriveStop => "WebDB".Z2Output.DriveMoving,
                     Standstill => "WebDB".Z2Output.StandStillControl,
                     MC => "WebDB".Z2Output.MC,
                     AXISModePos => "AXIS_Z2_Motion_V2_Festo_PtP_Drives_PN_DB".ModePos,
                     AXISEnableAxis => "AXIS_Z2_Motion_V2_Festo_PtP_Drives_PN_DB".EnableAxis,
                     AXISCancelTraversing => "AXIS_Z2_Motion_V2_Festo_PtP_Drives_PN_DB".CancelTraversing,
                     AXISIntermediateStop => "AXIS_Z2_Motion_V2_Festo_PtP_Drives_PN_DB".IntermediateStop,
                     AXISJog1 => "AXIS_Z2_Motion_V2_Festo_PtP_Drives_PN_DB".Jog1,
                     AXISJog2 => "AXIS_Z2_Motion_V2_Festo_PtP_Drives_PN_DB".Jog2,
                     AXISAckError => "AXIS_Z2_Motion_V2_Festo_PtP_Drives_PN_DB".AckError,
                     AXISExecuteMode => "AXIS_Z2_Motion_V2_Festo_PtP_Drives_PN_DB".ExecuteMode,
                     AXISPosition => "AXIS_Z2_Motion_V2_Festo_PtP_Drives_PN_DB".Position,
                     AXISVelocity => "AXIS_Z2_Motion_V2_Festo_PtP_Drives_PN_DB".Velocity,
                     AXISConfigEpos => "AXIS_Z2_Motion_V2_Festo_PtP_Drives_PN_DB".ConfigEPos,
                     FinishTask_Delay => "AXES_Positions_Delays".AXIS_Z2_Position_DelayIn,
                     ENO => #_w1);
   IF #_w1 THEN
       "AXIS_Z2_Motion_V2_Festo_PtP_Drives_PN_DB"(BaseSpeedValue := 20.0,   // "Festo_PtP_Drives_PN"
                               HardwareId := 309,
                               AxisEnabled => "WebDB".Z2Output.DriveEnabled,
                               AxisRef => "WebDB".Z2Output.HomingValid,
                               AxisWarn => "WebDB".Z2Output.Warning,
                               AxisError => "WebDB".Z2Output.Fault,
                               ActVelocity => "WebDB".Z2Output.ActualVelocity,
                               ActPosition => "WebDB".Z2Output.ActualPosition);
   END_IF;
END_REGION

REGION Network 5: AXIS Z2 CMMS
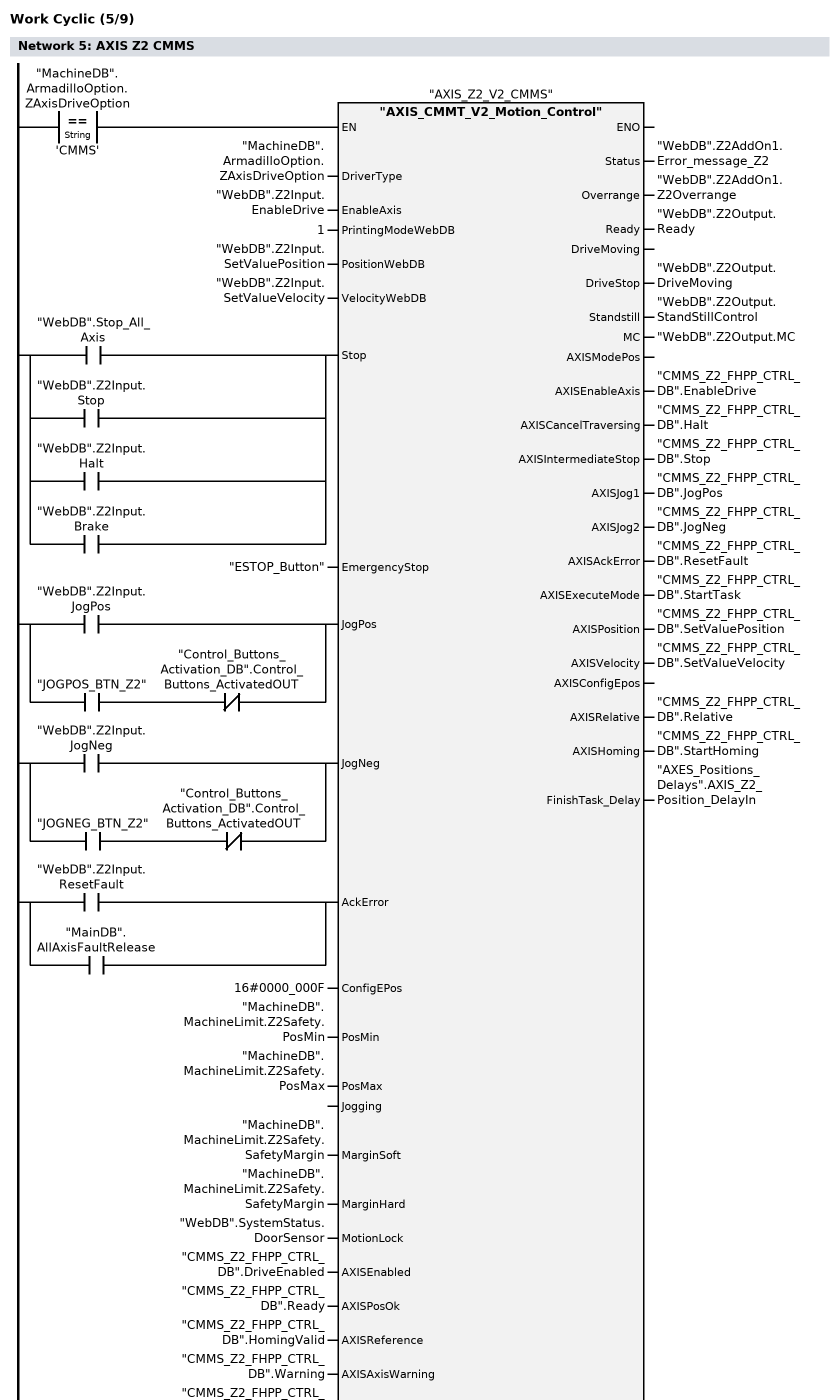
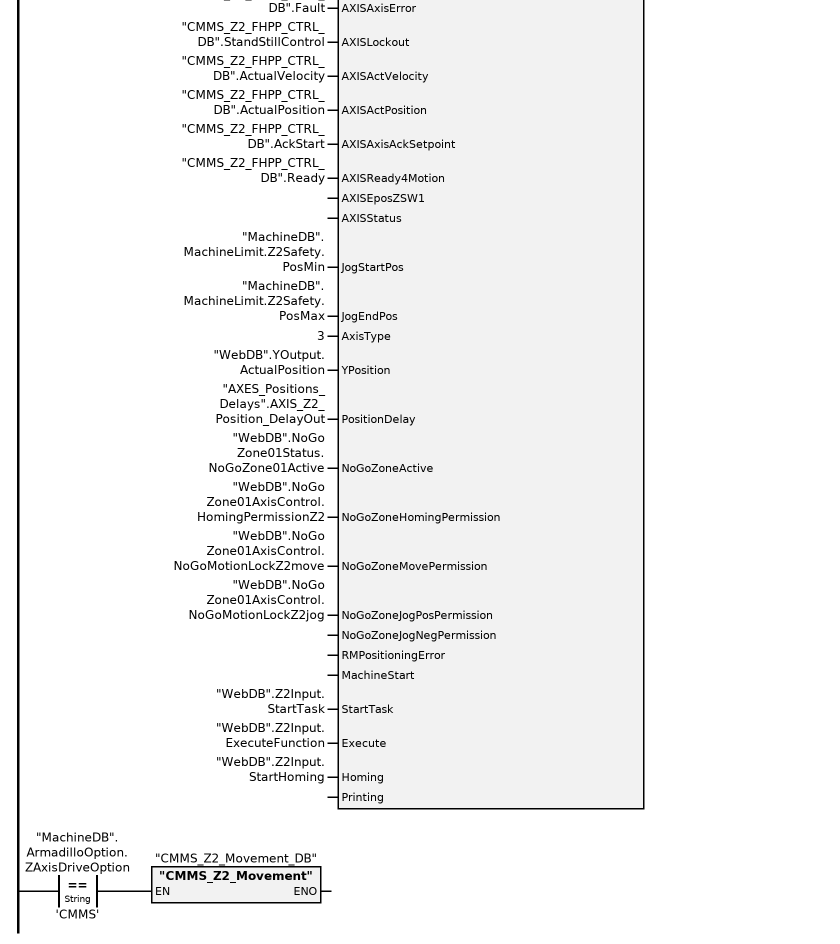
   RUNG wire#powerrail
      { S7_Templates := "SrcType := String" } EQ_Contact(in1 := "MachineDB".ArmadilloOption.ZAxisDriveOption, in2 := 'CMMS')
      "AXIS_Z2_V2_CMMS"(Stop := wire#w1, JogPos := wire#w2, JogNeg := wire#w3, AckError := wire#w4, DriverType := "MachineDB".ArmadilloOption.ZAxisDriveOption, EnableAxis := "WebDB".Z2Input.EnableDrive, PrintingModeWebDB := 1, PositionWebDB := "WebDB".Z2Input.SetValuePosition, VelocityWebDB := "WebDB".Z2Input.SetValueVelocity, EmergencyStop := "ESTOP_Button", ConfigEPos := 16#0000_000F, PosMin := "MachineDB".MachineLimit.Z2Safety.PosMin, PosMax := "MachineDB".MachineLimit.Z2Safety.PosMax, Jogging :=, MarginSoft := "MachineDB".MachineLimit.Z2Safety.SafetyMargin, MarginHard := "MachineDB".MachineLimit.Z2Safety.SafetyMargin, MotionLock := "WebDB".SystemStatus.DoorSensor, AXISEnabled := "CMMS_Z2_FHPP_CTRL_DB".DriveEnabled, AXISPosOk := "CMMS_Z2_FHPP_CTRL_DB".Ready, AXISReference := "CMMS_Z2_FHPP_CTRL_DB".HomingValid, AXISAxisWarning := "CMMS_Z2_FHPP_CTRL_DB".Warning, AXISAxisError := "CMMS_Z2_FHPP_CTRL_DB".Fault, AXISLockout := "CMMS_Z2_FHPP_CTRL_DB".StandStillControl, AXISActVelocity := "CMMS_Z2_FHPP_CTRL_DB".ActualVelocity, AXISActPosition := "CMMS_Z2_FHPP_CTRL_DB".ActualPosition, AXISAxisAckSetpoint := "CMMS_Z2_FHPP_CTRL_DB".AckStart, AXISReady4Motion := "CMMS_Z2_FHPP_CTRL_DB".Ready, AXISEposZSW1 :=, AXISStatus :=, JogStartPos := "MachineDB".MachineLimit.Z2Safety.PosMin, JogEndPos := "MachineDB".MachineLimit.Z2Safety.PosMax, AxisType := 3, YPosition := "WebDB".YOutput.ActualPosition, PositionDelay := "AXES_Positions_Delays".AXIS_Z2_Position_DelayOut, NoGoZoneActive := "WebDB".NoGoZone01Status.NoGoZone01Active, NoGoZoneHomingPermission := "WebDB".NoGoZone01AxisControl.HomingPermissionZ2, NoGoZoneMovePermission := "WebDB".NoGoZone01AxisControl.NoGoMotionLockZ2move, NoGoZoneJogPosPermission := "WebDB".NoGoZone01AxisControl.NoGoMotionLockZ2jog, NoGoZoneJogNegPermission :=, RMPositioningError :=, MachineStart :=, StartTask := "WebDB".Z2Input.StartTask, Execute := "WebDB".Z2Input.ExecuteFunction, Homing := "WebDB".Z2Input.StartHoming, Printing :=, Status => "WebDB".Z2AddOn1.Error_message_Z2, Overrange => "WebDB".Z2AddOn1.Z2Overrange, Ready => "WebDB".Z2Output.Ready, DriveMoving =>, DriveStop => "WebDB".Z2Output.DriveMoving, Standstill => "WebDB".Z2Output.StandStillControl, MC => "WebDB".Z2Output.MC, AXISModePos =>, AXISEnableAxis => "CMMS_Z2_FHPP_CTRL_DB".EnableDrive, AXISCancelTraversing => "CMMS_Z2_FHPP_CTRL_DB".Halt, AXISIntermediateStop => "CMMS_Z2_FHPP_CTRL_DB".Stop, AXISJog1 => "CMMS_Z2_FHPP_CTRL_DB".JogPos, AXISJog2 => "CMMS_Z2_FHPP_CTRL_DB".JogNeg, AXISAckError => "CMMS_Z2_FHPP_CTRL_DB".ResetFault, AXISExecuteMode => "CMMS_Z2_FHPP_CTRL_DB".StartTask, AXISPosition => "CMMS_Z2_FHPP_CTRL_DB".SetValuePosition, AXISVelocity => "CMMS_Z2_FHPP_CTRL_DB".SetValueVelocity, AXISConfigEpos =>, AXISRelative => "CMMS_Z2_FHPP_CTRL_DB".Relative, AXISHoming => "CMMS_Z2_FHPP_CTRL_DB".StartHoming, FinishTask_Delay => "AXES_Positions_Delays".AXIS_Z2_Position_DelayIn)
   END_RUNG
   RUNG wire#powerrail
      Contact( "WebDB".Stop_All_Axis )
   END_RUNG wire#w1
   RUNG wire#powerrail
      Contact( "WebDB".Z2Input.Stop )
   END_RUNG wire#w1
   RUNG wire#powerrail
      Contact( "WebDB".Z2Input.Halt )
   END_RUNG wire#w1
   RUNG wire#powerrail
      Contact( "WebDB".Z2Input.Brake )
   END_RUNG wire#w1
   RUNG wire#powerrail
      Contact( "WebDB".Z2Input.JogPos )
   END_RUNG wire#w2
   RUNG wire#powerrail
      Contact( "JOGPOS_BTN_Z2" )
      I_Contact( "Control_Buttons_Activation_DB".Control_Buttons_ActivatedOUT )
   END_RUNG wire#w2
   RUNG wire#powerrail
      Contact( "WebDB".Z2Input.JogNeg )
   END_RUNG wire#w3
   RUNG wire#powerrail
      Contact( "JOGNEG_BTN_Z2" )
      I_Contact( "Control_Buttons_Activation_DB".Control_Buttons_ActivatedOUT )
   END_RUNG wire#w3
   RUNG wire#powerrail
      Contact( "WebDB".Z2Input.ResetFault )
   END_RUNG wire#w4
   RUNG wire#powerrail
      Contact( "MainDB".AllAxisFaultRelease )
   END_RUNG wire#w4
   RUNG wire#powerrail
      { S7_Templates := "SrcType := String" } EQ_Contact(in1 := "MachineDB".ArmadilloOption.ZAxisDriveOption, in2 := 'CMMS')
      "CMMS_Z2_Movement_DB"()
   END_RUNG
   // the same network as SCL:
   IF "MachineDB".ArmadilloOption.ZAxisDriveOption = 'CMMS' THEN
       "AXIS_Z2_V2_CMMS"(DriverType := "MachineDB".ArmadilloOption.ZAxisDriveOption,   // "AXIS_CMMT_V2_Motion_Control"
                         EnableAxis := "WebDB".Z2Input.EnableDrive,
                         PrintingModeWebDB := 1,
                         PositionWebDB := "WebDB".Z2Input.SetValuePosition,
                         VelocityWebDB := "WebDB".Z2Input.SetValueVelocity,
                         Stop := "WebDB".Stop_All_Axis OR "WebDB".Z2Input.Stop OR "WebDB".Z2Input.Halt OR "WebDB".Z2Input.Brake,
                         EmergencyStop := "ESTOP_Button",
                         JogPos := "WebDB".Z2Input.JogPos OR ("JOGPOS_BTN_Z2" AND NOT "Control_Buttons_Activation_DB".Control_Buttons_ActivatedOUT),
                         JogNeg := "WebDB".Z2Input.JogNeg OR ("JOGNEG_BTN_Z2" AND NOT "Control_Buttons_Activation_DB".Control_Buttons_ActivatedOUT),
                         AckError := "WebDB".Z2Input.ResetFault OR "MainDB".AllAxisFaultRelease,
                         ConfigEPos := 16#0000_000F,
                         PosMin := "MachineDB".MachineLimit.Z2Safety.PosMin,
                         PosMax := "MachineDB".MachineLimit.Z2Safety.PosMax,
                         MarginSoft := "MachineDB".MachineLimit.Z2Safety.SafetyMargin,
                         MarginHard := "MachineDB".MachineLimit.Z2Safety.SafetyMargin,
                         MotionLock := "WebDB".SystemStatus.DoorSensor,
                         AXISEnabled := "CMMS_Z2_FHPP_CTRL_DB".DriveEnabled,
                         AXISPosOk := "CMMS_Z2_FHPP_CTRL_DB".Ready,
                         AXISReference := "CMMS_Z2_FHPP_CTRL_DB".HomingValid,
                         AXISAxisWarning := "CMMS_Z2_FHPP_CTRL_DB".Warning,
                         AXISAxisError := "CMMS_Z2_FHPP_CTRL_DB".Fault,
                         AXISLockout := "CMMS_Z2_FHPP_CTRL_DB".StandStillControl,
                         AXISActVelocity := "CMMS_Z2_FHPP_CTRL_DB".ActualVelocity,
                         AXISActPosition := "CMMS_Z2_FHPP_CTRL_DB".ActualPosition,
                         AXISAxisAckSetpoint := "CMMS_Z2_FHPP_CTRL_DB".AckStart,
                         AXISReady4Motion := "CMMS_Z2_FHPP_CTRL_DB".Ready,
                         JogStartPos := "MachineDB".MachineLimit.Z2Safety.PosMin,
                         JogEndPos := "MachineDB".MachineLimit.Z2Safety.PosMax,
                         AxisType := 3,
                         YPosition := "WebDB".YOutput.ActualPosition,
                         PositionDelay := "AXES_Positions_Delays".AXIS_Z2_Position_DelayOut,
                         NoGoZoneActive := "WebDB".NoGoZone01Status.NoGoZone01Active,
                         NoGoZoneHomingPermission := "WebDB".NoGoZone01AxisControl.HomingPermissionZ2,
                         NoGoZoneMovePermission := "WebDB".NoGoZone01AxisControl.NoGoMotionLockZ2move,
                         NoGoZoneJogPosPermission := "WebDB".NoGoZone01AxisControl.NoGoMotionLockZ2jog,
                         StartTask := "WebDB".Z2Input.StartTask,
                         Execute := "WebDB".Z2Input.ExecuteFunction,
                         Homing := "WebDB".Z2Input.StartHoming,
                         Status => "WebDB".Z2AddOn1.Error_message_Z2,
                         Overrange => "WebDB".Z2AddOn1.Z2Overrange,
                         Ready => "WebDB".Z2Output.Ready,
                         DriveStop => "WebDB".Z2Output.DriveMoving,
                         Standstill => "WebDB".Z2Output.StandStillControl,
                         MC => "WebDB".Z2Output.MC,
                         AXISEnableAxis => "CMMS_Z2_FHPP_CTRL_DB".EnableDrive,
                         AXISCancelTraversing => "CMMS_Z2_FHPP_CTRL_DB".Halt,
                         AXISIntermediateStop => "CMMS_Z2_FHPP_CTRL_DB".Stop,
                         AXISJog1 => "CMMS_Z2_FHPP_CTRL_DB".JogPos,
                         AXISJog2 => "CMMS_Z2_FHPP_CTRL_DB".JogNeg,
                         AXISAckError => "CMMS_Z2_FHPP_CTRL_DB".ResetFault,
                         AXISExecuteMode => "CMMS_Z2_FHPP_CTRL_DB".StartTask,
                         AXISPosition => "CMMS_Z2_FHPP_CTRL_DB".SetValuePosition,
                         AXISVelocity => "CMMS_Z2_FHPP_CTRL_DB".SetValueVelocity,
                         AXISRelative => "CMMS_Z2_FHPP_CTRL_DB".Relative,
                         AXISHoming => "CMMS_Z2_FHPP_CTRL_DB".StartHoming,
                         FinishTask_Delay => "AXES_Positions_Delays".AXIS_Z2_Position_DelayIn);
   END_IF;
   IF "MachineDB".ArmadilloOption.ZAxisDriveOption = 'CMMS' THEN
       "CMMS_Z2_Movement_DB"();   // "CMMS_Z2_Movement"
   END_IF;
END_REGION

REGION Network 6: AXIS Z2 Delays
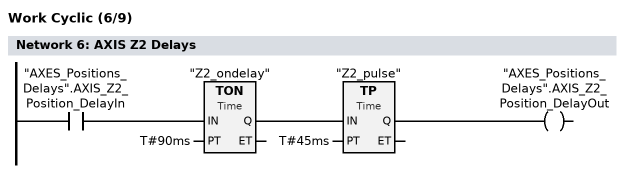
   RUNG wire#powerrail
      Contact( "AXES_Positions_Delays".AXIS_Z2_Position_DelayIn )
      { S7_Templates := "time_type := Time" } "Z2_ondelay".TON(pt := T#90ms, et =>)
      { S7_Templates := "time_type := Time" } "Z2_pulse".TP(pt := T#45ms, et =>)
      Coil( "AXES_Positions_Delays".AXIS_Z2_Position_DelayOut )
   END_RUNG
   // the same network as SCL:
   "Z2_ondelay".TON(IN := "AXES_Positions_Delays".AXIS_Z2_Position_DelayIn, PT := T#90ms);
   "Z2_pulse".TP(IN := "Z2_ondelay".Q, PT := T#45ms);
   "AXES_Positions_Delays".AXIS_Z2_Position_DelayOut := "Z2_pulse".Q;
END_REGION

REGION Network 7: AXIS X Control CMMT V2 To Update
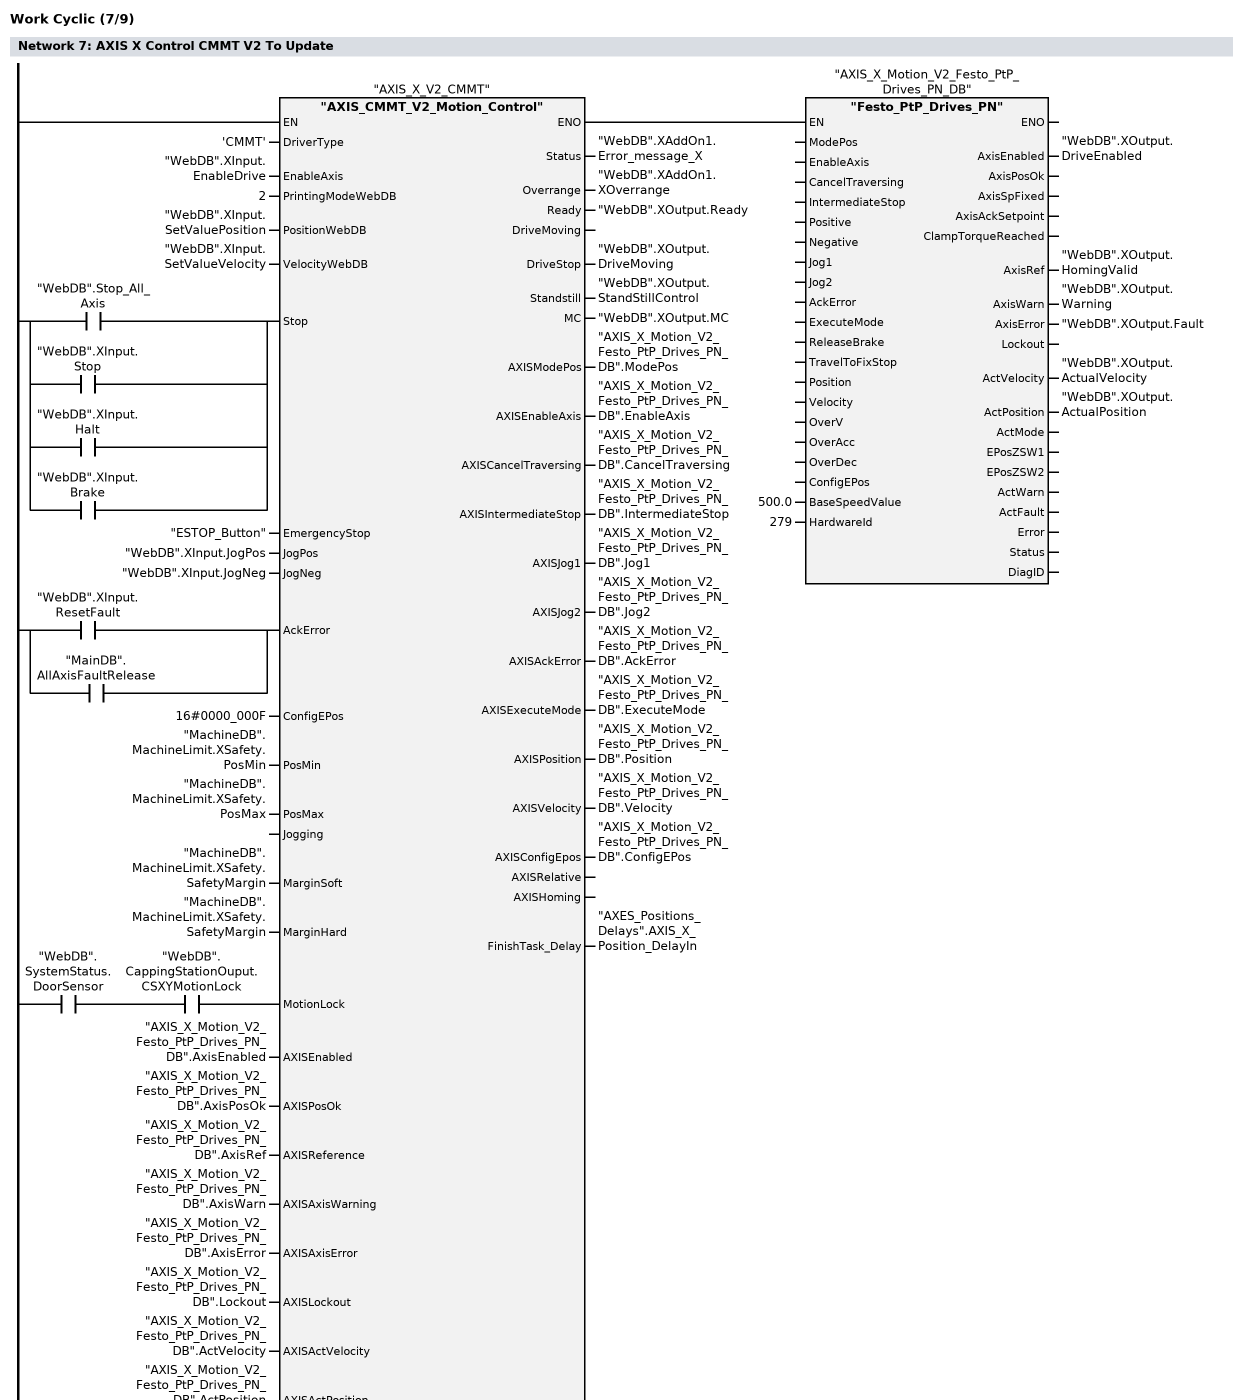
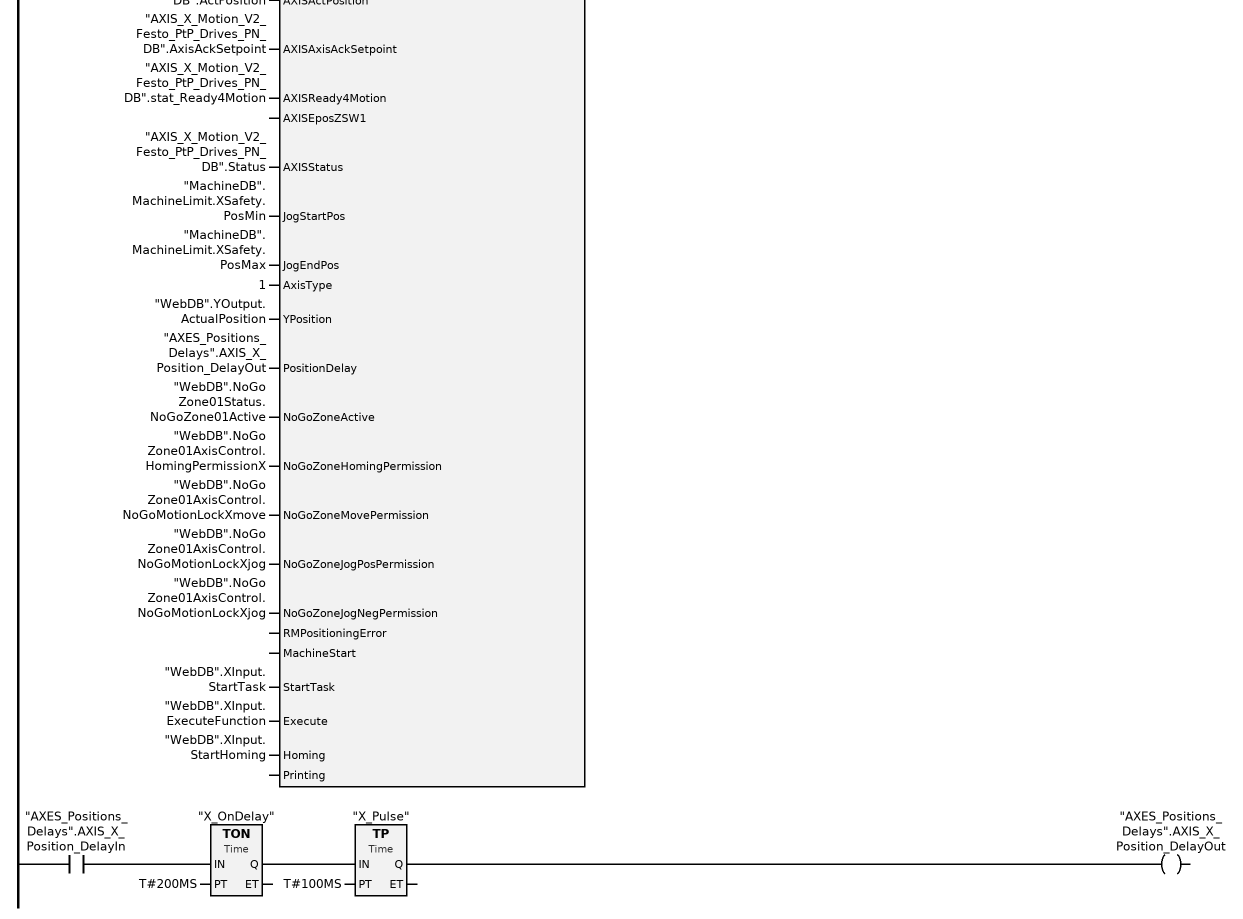
   RUNG wire#powerrail
      "AXIS_X_V2_CMMT"(Stop := wire#w1, AckError := wire#w2, MotionLock := wire#w3, DriverType := 'CMMT', EnableAxis := "WebDB".XInput.EnableDrive, PrintingModeWebDB := 2, PositionWebDB := "WebDB".XInput.SetValuePosition, VelocityWebDB := "WebDB".XInput.SetValueVelocity, EmergencyStop := "ESTOP_Button", JogPos := "WebDB".XInput.JogPos, JogNeg := "WebDB".XInput.JogNeg, ConfigEPos := 16#0000_000F, PosMin := "MachineDB".MachineLimit.XSafety.PosMin, PosMax := "MachineDB".MachineLimit.XSafety.PosMax, Jogging :=, MarginSoft := "MachineDB".MachineLimit.XSafety.SafetyMargin, MarginHard := "MachineDB".MachineLimit.XSafety.SafetyMargin, AXISEnabled := "AXIS_X_Motion_V2_Festo_PtP_Drives_PN_DB".AxisEnabled, AXISPosOk := "AXIS_X_Motion_V2_Festo_PtP_Drives_PN_DB".AxisPosOk, AXISReference := "AXIS_X_Motion_V2_Festo_PtP_Drives_PN_DB".AxisRef, AXISAxisWarning := "AXIS_X_Motion_V2_Festo_PtP_Drives_PN_DB".AxisWarn, AXISAxisError := "AXIS_X_Motion_V2_Festo_PtP_Drives_PN_DB".AxisError, AXISLockout := "AXIS_X_Motion_V2_Festo_PtP_Drives_PN_DB".Lockout, AXISActVelocity := "AXIS_X_Motion_V2_Festo_PtP_Drives_PN_DB".ActVelocity, AXISActPosition := "AXIS_X_Motion_V2_Festo_PtP_Drives_PN_DB".ActPosition, AXISAxisAckSetpoint := "AXIS_X_Motion_V2_Festo_PtP_Drives_PN_DB".AxisAckSetpoint, AXISReady4Motion := "AXIS_X_Motion_V2_Festo_PtP_Drives_PN_DB".stat_Ready4Motion, AXISEposZSW1 :=, AXISStatus := "AXIS_X_Motion_V2_Festo_PtP_Drives_PN_DB".Status, JogStartPos := "MachineDB".MachineLimit.XSafety.PosMin, JogEndPos := "MachineDB".MachineLimit.XSafety.PosMax, AxisType := 1, YPosition := "WebDB".YOutput.ActualPosition, PositionDelay := "AXES_Positions_Delays".AXIS_X_Position_DelayOut, NoGoZoneActive := "WebDB".NoGoZone01Status.NoGoZone01Active, NoGoZoneHomingPermission := "WebDB".NoGoZone01AxisControl.HomingPermissionX, NoGoZoneMovePermission := "WebDB".NoGoZone01AxisControl.NoGoMotionLockXmove, NoGoZoneJogPosPermission := "WebDB".NoGoZone01AxisControl.NoGoMotionLockXjog, NoGoZoneJogNegPermission := "WebDB".NoGoZone01AxisControl.NoGoMotionLockXjog, RMPositioningError :=, MachineStart :=, StartTask := "WebDB".XInput.StartTask, Execute := "WebDB".XInput.ExecuteFunction, Homing := "WebDB".XInput.StartHoming, Printing :=, Status => "WebDB".XAddOn1.Error_message_X, Overrange => "WebDB".XAddOn1.XOverrange, Ready => "WebDB".XOutput.Ready, DriveMoving =>, DriveStop => "WebDB".XOutput.DriveMoving, Standstill => "WebDB".XOutput.StandStillControl, MC => "WebDB".XOutput.MC, AXISModePos => "AXIS_X_Motion_V2_Festo_PtP_Drives_PN_DB".ModePos, AXISEnableAxis => "AXIS_X_Motion_V2_Festo_PtP_Drives_PN_DB".EnableAxis, AXISCancelTraversing => "AXIS_X_Motion_V2_Festo_PtP_Drives_PN_DB".CancelTraversing, AXISIntermediateStop => "AXIS_X_Motion_V2_Festo_PtP_Drives_PN_DB".IntermediateStop, AXISJog1 => "AXIS_X_Motion_V2_Festo_PtP_Drives_PN_DB".Jog1, AXISJog2 => "AXIS_X_Motion_V2_Festo_PtP_Drives_PN_DB".Jog2, AXISAckError => "AXIS_X_Motion_V2_Festo_PtP_Drives_PN_DB".AckError, AXISExecuteMode => "AXIS_X_Motion_V2_Festo_PtP_Drives_PN_DB".ExecuteMode, AXISPosition => "AXIS_X_Motion_V2_Festo_PtP_Drives_PN_DB".Position, AXISVelocity => "AXIS_X_Motion_V2_Festo_PtP_Drives_PN_DB".Velocity, AXISConfigEpos => "AXIS_X_Motion_V2_Festo_PtP_Drives_PN_DB".ConfigEPos, AXISRelative =>, AXISHoming =>, FinishTask_Delay => "AXES_Positions_Delays".AXIS_X_Position_DelayIn)
      "AXIS_X_Motion_V2_Festo_PtP_Drives_PN_DB"(ModePos :=, EnableAxis :=, CancelTraversing :=, IntermediateStop :=, Positive :=, Negative :=, Jog1 :=, Jog2 :=, AckError :=, ExecuteMode :=, ReleaseBrake :=, TravelToFixStop :=, Position :=, Velocity :=, OverV :=, OverAcc :=, OverDec :=, ConfigEPos :=, BaseSpeedValue := 500.0, HardwareId := 279, AxisEnabled => "WebDB".XOutput.DriveEnabled, AxisPosOk =>, AxisSpFixed =>, AxisAckSetpoint =>, ClampTorqueReached =>, AxisRef => "WebDB".XOutput.HomingValid, AxisWarn => "WebDB".XOutput.Warning, AxisError => "WebDB".XOutput.Fault, Lockout =>, ActVelocity => "WebDB".XOutput.ActualVelocity, ActPosition => "WebDB".XOutput.ActualPosition, ActMode =>, EPosZSW1 =>, EPosZSW2 =>, ActWarn =>, ActFault =>, Error =>, Status =>, DiagID =>)
   END_RUNG
   RUNG wire#powerrail
      Contact( "WebDB".Stop_All_Axis )
   END_RUNG wire#w1
   RUNG wire#powerrail
      Contact( "WebDB".XInput.Stop )
   END_RUNG wire#w1
   RUNG wire#powerrail
      Contact( "WebDB".XInput.Halt )
   END_RUNG wire#w1
   RUNG wire#powerrail
      Contact( "WebDB".XInput.Brake )
   END_RUNG wire#w1
   RUNG wire#powerrail
      Contact( "WebDB".XInput.ResetFault )
   END_RUNG wire#w2
   RUNG wire#powerrail
      Contact( "MainDB".AllAxisFaultRelease )
   END_RUNG wire#w2
   RUNG wire#powerrail
      Contact( "WebDB".SystemStatus.DoorSensor )
      Contact( "WebDB".CappingStationOuput.CSXYMotionLock )
   END_RUNG wire#w3
   RUNG wire#powerrail
      Contact( "AXES_Positions_Delays".AXIS_X_Position_DelayIn )
      { S7_Templates := "time_type := Time" } "X_OnDelay".TON(pt := T#200MS, et =>)
      { S7_Templates := "time_type := Time" } "X_Pulse".TP(pt := T#100MS, et =>)
      Coil( "AXES_Positions_Delays".AXIS_X_Position_DelayOut )
   END_RUNG
   // the same network as SCL:
   "AXIS_X_V2_CMMT"(DriverType := 'CMMT',   // "AXIS_CMMT_V2_Motion_Control"
                    EnableAxis := "WebDB".XInput.EnableDrive,
                    PrintingModeWebDB := 2,
                    PositionWebDB := "WebDB".XInput.SetValuePosition,
                    VelocityWebDB := "WebDB".XInput.SetValueVelocity,
                    Stop := "WebDB".Stop_All_Axis OR "WebDB".XInput.Stop OR "WebDB".XInput.Halt OR "WebDB".XInput.Brake,
                    EmergencyStop := "ESTOP_Button",
                    JogPos := "WebDB".XInput.JogPos,
                    JogNeg := "WebDB".XInput.JogNeg,
                    AckError := "WebDB".XInput.ResetFault OR "MainDB".AllAxisFaultRelease,
                    ConfigEPos := 16#0000_000F,
                    PosMin := "MachineDB".MachineLimit.XSafety.PosMin,
                    PosMax := "MachineDB".MachineLimit.XSafety.PosMax,
                    MarginSoft := "MachineDB".MachineLimit.XSafety.SafetyMargin,
                    MarginHard := "MachineDB".MachineLimit.XSafety.SafetyMargin,
                    MotionLock := "WebDB".SystemStatus.DoorSensor AND "WebDB".CappingStationOuput.CSXYMotionLock,
                    AXISEnabled := "AXIS_X_Motion_V2_Festo_PtP_Drives_PN_DB".AxisEnabled,
                    AXISPosOk := "AXIS_X_Motion_V2_Festo_PtP_Drives_PN_DB".AxisPosOk,
                    AXISReference := "AXIS_X_Motion_V2_Festo_PtP_Drives_PN_DB".AxisRef,
                    AXISAxisWarning := "AXIS_X_Motion_V2_Festo_PtP_Drives_PN_DB".AxisWarn,
                    AXISAxisError := "AXIS_X_Motion_V2_Festo_PtP_Drives_PN_DB".AxisError,
                    AXISLockout := "AXIS_X_Motion_V2_Festo_PtP_Drives_PN_DB".Lockout,
                    AXISActVelocity := "AXIS_X_Motion_V2_Festo_PtP_Drives_PN_DB".ActVelocity,
                    AXISActPosition := "AXIS_X_Motion_V2_Festo_PtP_Drives_PN_DB".ActPosition,
                    AXISAxisAckSetpoint := "AXIS_X_Motion_V2_Festo_PtP_Drives_PN_DB".AxisAckSetpoint,
                    AXISReady4Motion := "AXIS_X_Motion_V2_Festo_PtP_Drives_PN_DB".stat_Ready4Motion,
                    AXISStatus := "AXIS_X_Motion_V2_Festo_PtP_Drives_PN_DB".Status,
                    JogStartPos := "MachineDB".MachineLimit.XSafety.PosMin,
                    JogEndPos := "MachineDB".MachineLimit.XSafety.PosMax,
                    AxisType := 1,
                    YPosition := "WebDB".YOutput.ActualPosition,
                    PositionDelay := "AXES_Positions_Delays".AXIS_X_Position_DelayOut,
                    NoGoZoneActive := "WebDB".NoGoZone01Status.NoGoZone01Active,
                    NoGoZoneHomingPermission := "WebDB".NoGoZone01AxisControl.HomingPermissionX,
                    NoGoZoneMovePermission := "WebDB".NoGoZone01AxisControl.NoGoMotionLockXmove,
                    NoGoZoneJogPosPermission := "WebDB".NoGoZone01AxisControl.NoGoMotionLockXjog,
                    NoGoZoneJogNegPermission := "WebDB".NoGoZone01AxisControl.NoGoMotionLockXjog,
                    StartTask := "WebDB".XInput.StartTask,
                    Execute := "WebDB".XInput.ExecuteFunction,
                    Homing := "WebDB".XInput.StartHoming,
                    Status => "WebDB".XAddOn1.Error_message_X,
                    Overrange => "WebDB".XAddOn1.XOverrange,
                    Ready => "WebDB".XOutput.Ready,
                    DriveStop => "WebDB".XOutput.DriveMoving,
                    Standstill => "WebDB".XOutput.StandStillControl,
                    MC => "WebDB".XOutput.MC,
                    AXISModePos => "AXIS_X_Motion_V2_Festo_PtP_Drives_PN_DB".ModePos,
                    AXISEnableAxis => "AXIS_X_Motion_V2_Festo_PtP_Drives_PN_DB".EnableAxis,
                    AXISCancelTraversing => "AXIS_X_Motion_V2_Festo_PtP_Drives_PN_DB".CancelTraversing,
                    AXISIntermediateStop => "AXIS_X_Motion_V2_Festo_PtP_Drives_PN_DB".IntermediateStop,
                    AXISJog1 => "AXIS_X_Motion_V2_Festo_PtP_Drives_PN_DB".Jog1,
                    AXISJog2 => "AXIS_X_Motion_V2_Festo_PtP_Drives_PN_DB".Jog2,
                    AXISAckError => "AXIS_X_Motion_V2_Festo_PtP_Drives_PN_DB".AckError,
                    AXISExecuteMode => "AXIS_X_Motion_V2_Festo_PtP_Drives_PN_DB".ExecuteMode,
                    AXISPosition => "AXIS_X_Motion_V2_Festo_PtP_Drives_PN_DB".Position,
                    AXISVelocity => "AXIS_X_Motion_V2_Festo_PtP_Drives_PN_DB".Velocity,
                    AXISConfigEpos => "AXIS_X_Motion_V2_Festo_PtP_Drives_PN_DB".ConfigEPos,
                    FinishTask_Delay => "AXES_Positions_Delays".AXIS_X_Position_DelayIn,
                    ENO => #_w1);
   IF #_w1 THEN
       "AXIS_X_Motion_V2_Festo_PtP_Drives_PN_DB"(BaseSpeedValue := 500.0,   // "Festo_PtP_Drives_PN"
                               HardwareId := 279,
                               AxisEnabled => "WebDB".XOutput.DriveEnabled,
                               AxisRef => "WebDB".XOutput.HomingValid,
                               AxisWarn => "WebDB".XOutput.Warning,
                               AxisError => "WebDB".XOutput.Fault,
                               ActVelocity => "WebDB".XOutput.ActualVelocity,
                               ActPosition => "WebDB".XOutput.ActualPosition);
   END_IF;
   "X_OnDelay".TON(IN := "AXES_Positions_Delays".AXIS_X_Position_DelayIn, PT := T#200MS);
   "X_Pulse".TP(IN := "X_OnDelay".Q, PT := T#100MS);
   "AXES_Positions_Delays".AXIS_X_Position_DelayOut := "X_Pulse".Q;
END_REGION

REGION Network 8: AXIS Y Control CMMT V2 To Update
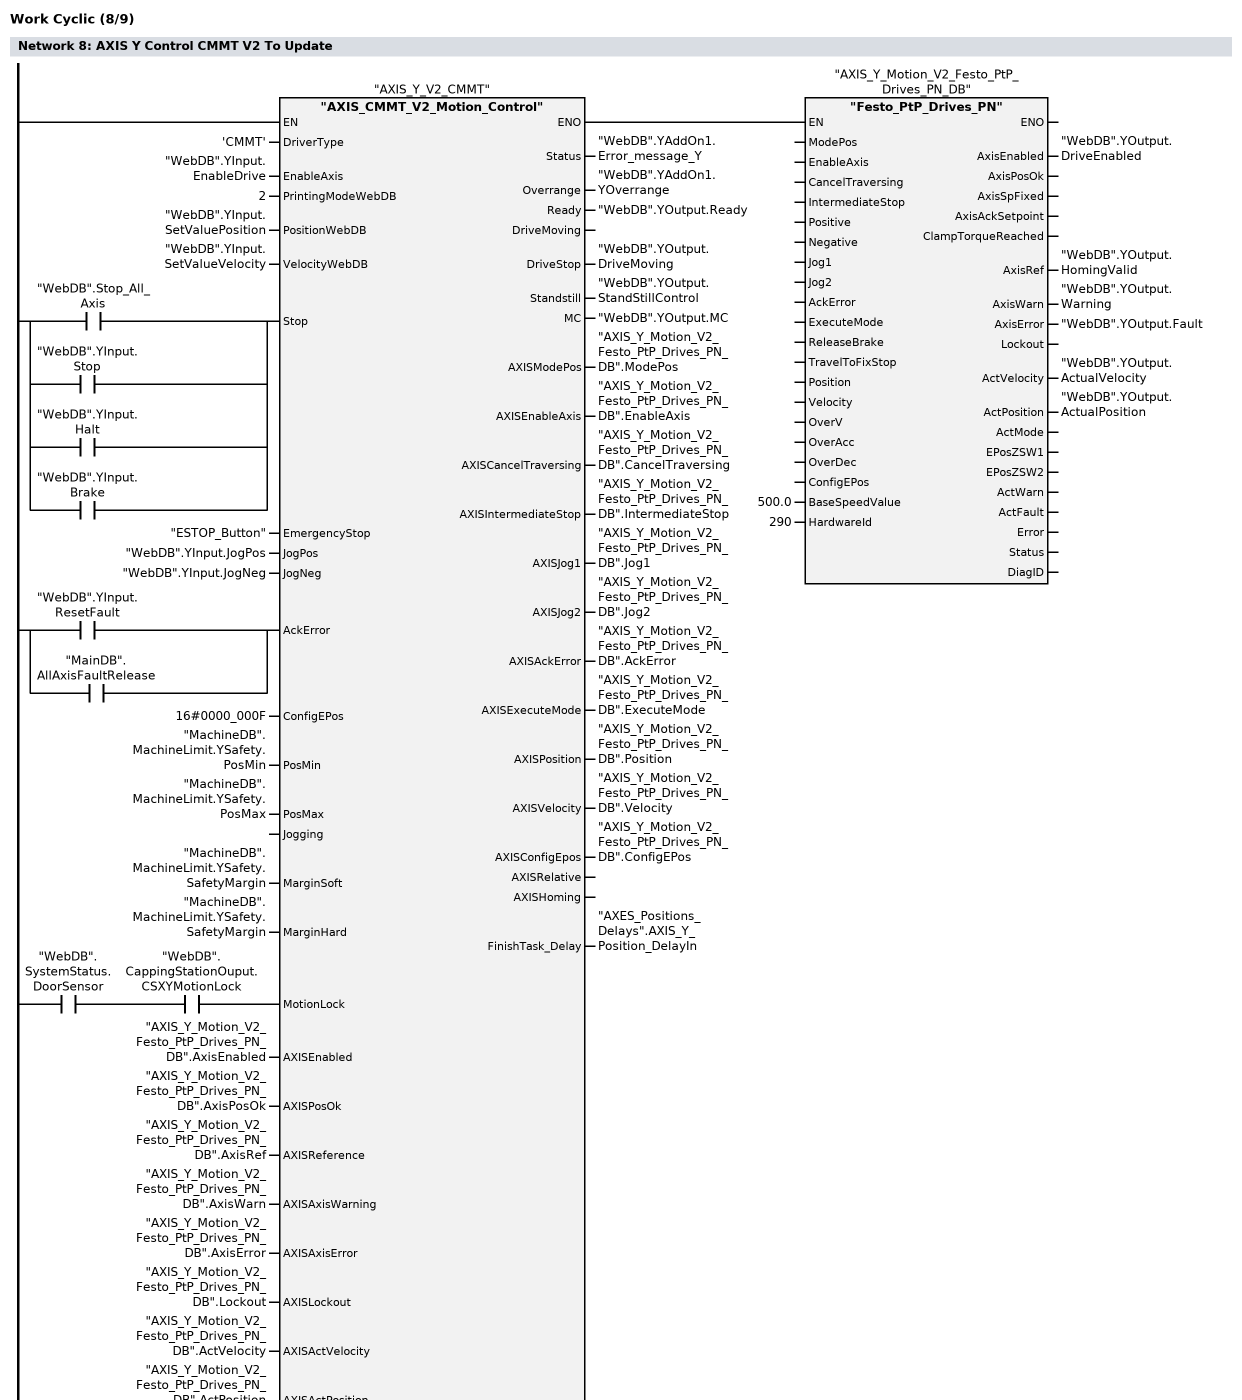
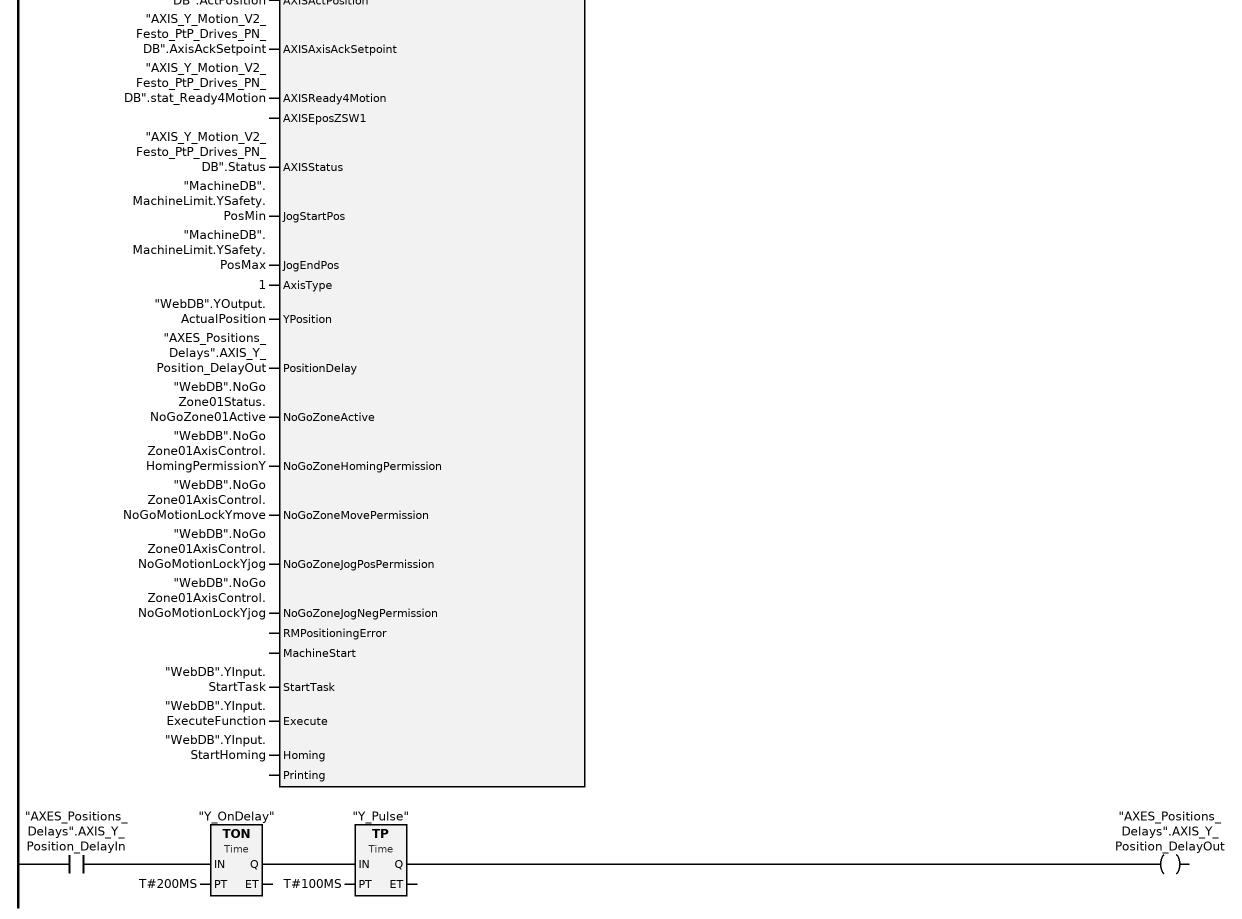
   RUNG wire#powerrail
      "AXIS_Y_V2_CMMT"(Stop := wire#w1, AckError := wire#w2, MotionLock := wire#w3, DriverType := 'CMMT', EnableAxis := "WebDB".YInput.EnableDrive, PrintingModeWebDB := 2, PositionWebDB := "WebDB".YInput.SetValuePosition, VelocityWebDB := "WebDB".YInput.SetValueVelocity, EmergencyStop := "ESTOP_Button", JogPos := "WebDB".YInput.JogPos, JogNeg := "WebDB".YInput.JogNeg, ConfigEPos := 16#0000_000F, PosMin := "MachineDB".MachineLimit.YSafety.PosMin, PosMax := "MachineDB".MachineLimit.YSafety.PosMax, Jogging :=, MarginSoft := "MachineDB".MachineLimit.YSafety.SafetyMargin, MarginHard := "MachineDB".MachineLimit.YSafety.SafetyMargin, AXISEnabled := "AXIS_Y_Motion_V2_Festo_PtP_Drives_PN_DB".AxisEnabled, AXISPosOk := "AXIS_Y_Motion_V2_Festo_PtP_Drives_PN_DB".AxisPosOk, AXISReference := "AXIS_Y_Motion_V2_Festo_PtP_Drives_PN_DB".AxisRef, AXISAxisWarning := "AXIS_Y_Motion_V2_Festo_PtP_Drives_PN_DB".AxisWarn, AXISAxisError := "AXIS_Y_Motion_V2_Festo_PtP_Drives_PN_DB".AxisError, AXISLockout := "AXIS_Y_Motion_V2_Festo_PtP_Drives_PN_DB".Lockout, AXISActVelocity := "AXIS_Y_Motion_V2_Festo_PtP_Drives_PN_DB".ActVelocity, AXISActPosition := "AXIS_Y_Motion_V2_Festo_PtP_Drives_PN_DB".ActPosition, AXISAxisAckSetpoint := "AXIS_Y_Motion_V2_Festo_PtP_Drives_PN_DB".AxisAckSetpoint, AXISReady4Motion := "AXIS_Y_Motion_V2_Festo_PtP_Drives_PN_DB".stat_Ready4Motion, AXISEposZSW1 :=, AXISStatus := "AXIS_Y_Motion_V2_Festo_PtP_Drives_PN_DB".Status, JogStartPos := "MachineDB".MachineLimit.YSafety.PosMin, JogEndPos := "MachineDB".MachineLimit.YSafety.PosMax, AxisType := 1, YPosition := "WebDB".YOutput.ActualPosition, PositionDelay := "AXES_Positions_Delays".AXIS_Y_Position_DelayOut, NoGoZoneActive := "WebDB".NoGoZone01Status.NoGoZone01Active, NoGoZoneHomingPermission := "WebDB".NoGoZone01AxisControl.HomingPermissionY, NoGoZoneMovePermission := "WebDB".NoGoZone01AxisControl.NoGoMotionLockYmove, NoGoZoneJogPosPermission := "WebDB".NoGoZone01AxisControl.NoGoMotionLockYjog, NoGoZoneJogNegPermission := "WebDB".NoGoZone01AxisControl.NoGoMotionLockYjog, RMPositioningError :=, MachineStart :=, StartTask := "WebDB".YInput.StartTask, Execute := "WebDB".YInput.ExecuteFunction, Homing := "WebDB".YInput.StartHoming, Printing :=, Status => "WebDB".YAddOn1.Error_message_Y, Overrange => "WebDB".YAddOn1.YOverrange, Ready => "WebDB".YOutput.Ready, DriveMoving =>, DriveStop => "WebDB".YOutput.DriveMoving, Standstill => "WebDB".YOutput.StandStillControl, MC => "WebDB".YOutput.MC, AXISModePos => "AXIS_Y_Motion_V2_Festo_PtP_Drives_PN_DB".ModePos, AXISEnableAxis => "AXIS_Y_Motion_V2_Festo_PtP_Drives_PN_DB".EnableAxis, AXISCancelTraversing => "AXIS_Y_Motion_V2_Festo_PtP_Drives_PN_DB".CancelTraversing, AXISIntermediateStop => "AXIS_Y_Motion_V2_Festo_PtP_Drives_PN_DB".IntermediateStop, AXISJog1 => "AXIS_Y_Motion_V2_Festo_PtP_Drives_PN_DB".Jog1, AXISJog2 => "AXIS_Y_Motion_V2_Festo_PtP_Drives_PN_DB".Jog2, AXISAckError => "AXIS_Y_Motion_V2_Festo_PtP_Drives_PN_DB".AckError, AXISExecuteMode => "AXIS_Y_Motion_V2_Festo_PtP_Drives_PN_DB".ExecuteMode, AXISPosition => "AXIS_Y_Motion_V2_Festo_PtP_Drives_PN_DB".Position, AXISVelocity => "AXIS_Y_Motion_V2_Festo_PtP_Drives_PN_DB".Velocity, AXISConfigEpos => "AXIS_Y_Motion_V2_Festo_PtP_Drives_PN_DB".ConfigEPos, AXISRelative =>, AXISHoming =>, FinishTask_Delay => "AXES_Positions_Delays".AXIS_Y_Position_DelayIn)
      "AXIS_Y_Motion_V2_Festo_PtP_Drives_PN_DB"(ModePos :=, EnableAxis :=, CancelTraversing :=, IntermediateStop :=, Positive :=, Negative :=, Jog1 :=, Jog2 :=, AckError :=, ExecuteMode :=, ReleaseBrake :=, TravelToFixStop :=, Position :=, Velocity :=, OverV :=, OverAcc :=, OverDec :=, ConfigEPos :=, BaseSpeedValue := 500.0, HardwareId := 290, AxisEnabled => "WebDB".YOutput.DriveEnabled, AxisPosOk =>, AxisSpFixed =>, AxisAckSetpoint =>, ClampTorqueReached =>, AxisRef => "WebDB".YOutput.HomingValid, AxisWarn => "WebDB".YOutput.Warning, AxisError => "WebDB".YOutput.Fault, Lockout =>, ActVelocity => "WebDB".YOutput.ActualVelocity, ActPosition => "WebDB".YOutput.ActualPosition, ActMode =>, EPosZSW1 =>, EPosZSW2 =>, ActWarn =>, ActFault =>, Error =>, Status =>, DiagID =>)
   END_RUNG
   RUNG wire#powerrail
      Contact( "WebDB".Stop_All_Axis )
   END_RUNG wire#w1
   RUNG wire#powerrail
      Contact( "WebDB".YInput.Stop )
   END_RUNG wire#w1
   RUNG wire#powerrail
      Contact( "WebDB".YInput.Halt )
   END_RUNG wire#w1
   RUNG wire#powerrail
      Contact( "WebDB".YInput.Brake )
   END_RUNG wire#w1
   RUNG wire#powerrail
      Contact( "WebDB".YInput.ResetFault )
   END_RUNG wire#w2
   RUNG wire#powerrail
      Contact( "MainDB".AllAxisFaultRelease )
   END_RUNG wire#w2
   RUNG wire#powerrail
      Contact( "WebDB".SystemStatus.DoorSensor )
      Contact( "WebDB".CappingStationOuput.CSXYMotionLock )
   END_RUNG wire#w3
   RUNG wire#powerrail
      Contact( "AXES_Positions_Delays".AXIS_Y_Position_DelayIn )
      { S7_Templates := "time_type := Time" } "Y_OnDelay".TON(pt := T#200MS, et =>)
      { S7_Templates := "time_type := Time" } "Y_Pulse".TP(pt := T#100MS, et =>)
      Coil( "AXES_Positions_Delays".AXIS_Y_Position_DelayOut )
   END_RUNG
   // the same network as SCL:
   "AXIS_Y_V2_CMMT"(DriverType := 'CMMT',   // "AXIS_CMMT_V2_Motion_Control"
                    EnableAxis := "WebDB".YInput.EnableDrive,
                    PrintingModeWebDB := 2,
                    PositionWebDB := "WebDB".YInput.SetValuePosition,
                    VelocityWebDB := "WebDB".YInput.SetValueVelocity,
                    Stop := "WebDB".Stop_All_Axis OR "WebDB".YInput.Stop OR "WebDB".YInput.Halt OR "WebDB".YInput.Brake,
                    EmergencyStop := "ESTOP_Button",
                    JogPos := "WebDB".YInput.JogPos,
                    JogNeg := "WebDB".YInput.JogNeg,
                    AckError := "WebDB".YInput.ResetFault OR "MainDB".AllAxisFaultRelease,
                    ConfigEPos := 16#0000_000F,
                    PosMin := "MachineDB".MachineLimit.YSafety.PosMin,
                    PosMax := "MachineDB".MachineLimit.YSafety.PosMax,
                    MarginSoft := "MachineDB".MachineLimit.YSafety.SafetyMargin,
                    MarginHard := "MachineDB".MachineLimit.YSafety.SafetyMargin,
                    MotionLock := "WebDB".SystemStatus.DoorSensor AND "WebDB".CappingStationOuput.CSXYMotionLock,
                    AXISEnabled := "AXIS_Y_Motion_V2_Festo_PtP_Drives_PN_DB".AxisEnabled,
                    AXISPosOk := "AXIS_Y_Motion_V2_Festo_PtP_Drives_PN_DB".AxisPosOk,
                    AXISReference := "AXIS_Y_Motion_V2_Festo_PtP_Drives_PN_DB".AxisRef,
                    AXISAxisWarning := "AXIS_Y_Motion_V2_Festo_PtP_Drives_PN_DB".AxisWarn,
                    AXISAxisError := "AXIS_Y_Motion_V2_Festo_PtP_Drives_PN_DB".AxisError,
                    AXISLockout := "AXIS_Y_Motion_V2_Festo_PtP_Drives_PN_DB".Lockout,
                    AXISActVelocity := "AXIS_Y_Motion_V2_Festo_PtP_Drives_PN_DB".ActVelocity,
                    AXISActPosition := "AXIS_Y_Motion_V2_Festo_PtP_Drives_PN_DB".ActPosition,
                    AXISAxisAckSetpoint := "AXIS_Y_Motion_V2_Festo_PtP_Drives_PN_DB".AxisAckSetpoint,
                    AXISReady4Motion := "AXIS_Y_Motion_V2_Festo_PtP_Drives_PN_DB".stat_Ready4Motion,
                    AXISStatus := "AXIS_Y_Motion_V2_Festo_PtP_Drives_PN_DB".Status,
                    JogStartPos := "MachineDB".MachineLimit.YSafety.PosMin,
                    JogEndPos := "MachineDB".MachineLimit.YSafety.PosMax,
                    AxisType := 1,
                    YPosition := "WebDB".YOutput.ActualPosition,
                    PositionDelay := "AXES_Positions_Delays".AXIS_Y_Position_DelayOut,
                    NoGoZoneActive := "WebDB".NoGoZone01Status.NoGoZone01Active,
                    NoGoZoneHomingPermission := "WebDB".NoGoZone01AxisControl.HomingPermissionY,
                    NoGoZoneMovePermission := "WebDB".NoGoZone01AxisControl.NoGoMotionLockYmove,
                    NoGoZoneJogPosPermission := "WebDB".NoGoZone01AxisControl.NoGoMotionLockYjog,
                    NoGoZoneJogNegPermission := "WebDB".NoGoZone01AxisControl.NoGoMotionLockYjog,
                    StartTask := "WebDB".YInput.StartTask,
                    Execute := "WebDB".YInput.ExecuteFunction,
                    Homing := "WebDB".YInput.StartHoming,
                    Status => "WebDB".YAddOn1.Error_message_Y,
                    Overrange => "WebDB".YAddOn1.YOverrange,
                    Ready => "WebDB".YOutput.Ready,
                    DriveStop => "WebDB".YOutput.DriveMoving,
                    Standstill => "WebDB".YOutput.StandStillControl,
                    MC => "WebDB".YOutput.MC,
                    AXISModePos => "AXIS_Y_Motion_V2_Festo_PtP_Drives_PN_DB".ModePos,
                    AXISEnableAxis => "AXIS_Y_Motion_V2_Festo_PtP_Drives_PN_DB".EnableAxis,
                    AXISCancelTraversing => "AXIS_Y_Motion_V2_Festo_PtP_Drives_PN_DB".CancelTraversing,
                    AXISIntermediateStop => "AXIS_Y_Motion_V2_Festo_PtP_Drives_PN_DB".IntermediateStop,
                    AXISJog1 => "AXIS_Y_Motion_V2_Festo_PtP_Drives_PN_DB".Jog1,
                    AXISJog2 => "AXIS_Y_Motion_V2_Festo_PtP_Drives_PN_DB".Jog2,
                    AXISAckError => "AXIS_Y_Motion_V2_Festo_PtP_Drives_PN_DB".AckError,
                    AXISExecuteMode => "AXIS_Y_Motion_V2_Festo_PtP_Drives_PN_DB".ExecuteMode,
                    AXISPosition => "AXIS_Y_Motion_V2_Festo_PtP_Drives_PN_DB".Position,
                    AXISVelocity => "AXIS_Y_Motion_V2_Festo_PtP_Drives_PN_DB".Velocity,
                    AXISConfigEpos => "AXIS_Y_Motion_V2_Festo_PtP_Drives_PN_DB".ConfigEPos,
                    FinishTask_Delay => "AXES_Positions_Delays".AXIS_Y_Position_DelayIn,
                    ENO => #_w1);
   IF #_w1 THEN
       "AXIS_Y_Motion_V2_Festo_PtP_Drives_PN_DB"(BaseSpeedValue := 500.0,   // "Festo_PtP_Drives_PN"
                               HardwareId := 290,
                               AxisEnabled => "WebDB".YOutput.DriveEnabled,
                               AxisRef => "WebDB".YOutput.HomingValid,
                               AxisWarn => "WebDB".YOutput.Warning,
                               AxisError => "WebDB".YOutput.Fault,
                               ActVelocity => "WebDB".YOutput.ActualVelocity,
                               ActPosition => "WebDB".YOutput.ActualPosition);
   END_IF;
   "Y_OnDelay".TON(IN := "AXES_Positions_Delays".AXIS_Y_Position_DelayIn, PT := T#200MS);
   "Y_Pulse".TP(IN := "Y_OnDelay".Q, PT := T#100MS);
   "AXES_Positions_Delays".AXIS_Y_Position_DelayOut := "Y_Pulse".Q;
END_REGION

REGION Network 9: Roller V3
   // The RollerV3 block already writes the roller speed and direction to the technology object. This means that the outputs are no longer needed.
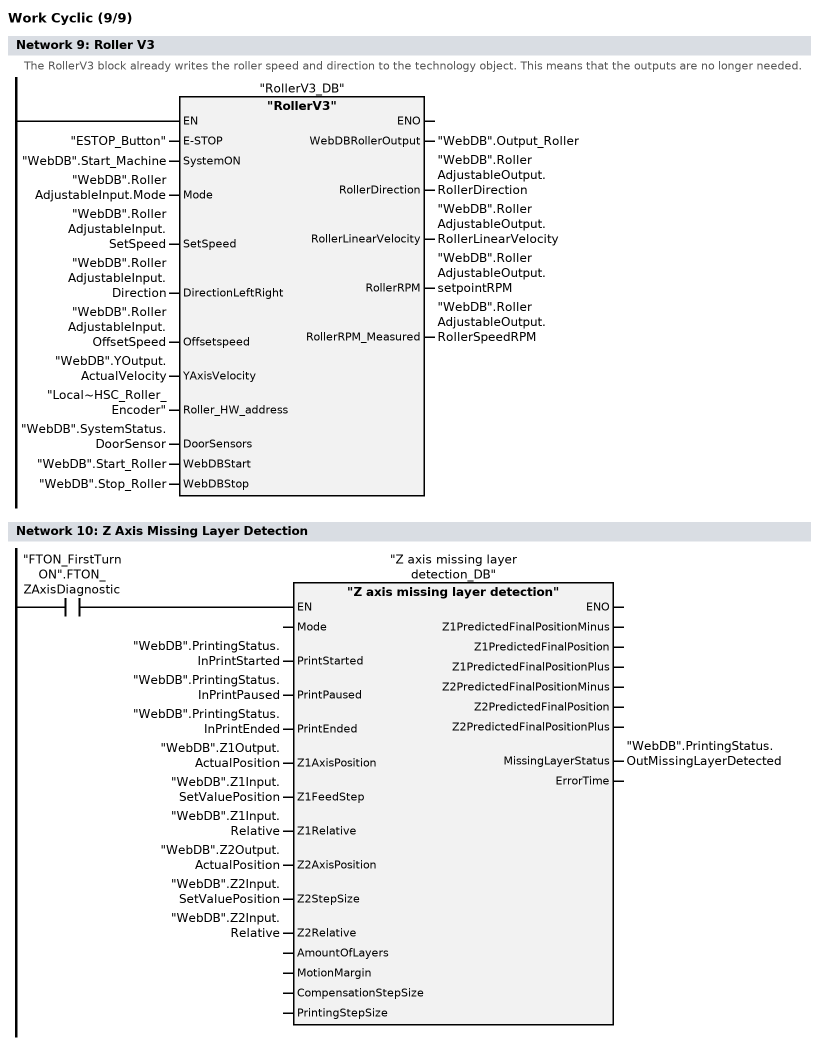
   RUNG wire#powerrail
      "RollerV3_DB"("E-STOP" := "ESTOP_Button", SystemON := "WebDB".Start_Machine, Mode := "WebDB".RollerAdjustableInput.Mode, SetSpeed := "WebDB".RollerAdjustableInput.SetSpeed, DirectionLeftRight := "WebDB".RollerAdjustableInput.Direction, Offsetspeed := "WebDB".RollerAdjustableInput.OffsetSpeed, YAxisVelocity := "WebDB".YOutput.ActualVelocity, Roller_HW_address := "Local~HSC_Roller_Encoder", DoorSensors := "WebDB".SystemStatus.DoorSensor, WebDBStart := "WebDB".Start_Roller, WebDBStop := "WebDB".Stop_Roller, WebDBRollerOutput => "WebDB".Output_Roller, RollerDirection => "WebDB".RollerAdjustableOutput.RollerDirection, RollerLinearVelocity => "WebDB".RollerAdjustableOutput.RollerLinearVelocity, RollerRPM => "WebDB".RollerAdjustableOutput.setpointRPM, RollerRPM_Measured => "WebDB".RollerAdjustableOutput.RollerSpeedRPM)
   END_RUNG
   // the same network as SCL:
   "RollerV3_DB"("E-STOP" := "ESTOP_Button",   // "RollerV3"
                 SystemON := "WebDB".Start_Machine,
                 Mode := "WebDB".RollerAdjustableInput.Mode,
                 SetSpeed := "WebDB".RollerAdjustableInput.SetSpeed,
                 DirectionLeftRight := "WebDB".RollerAdjustableInput.Direction,
                 Offsetspeed := "WebDB".RollerAdjustableInput.OffsetSpeed,
                 YAxisVelocity := "WebDB".YOutput.ActualVelocity,
                 Roller_HW_address := "Local~HSC_Roller_Encoder",
                 DoorSensors := "WebDB".SystemStatus.DoorSensor,
                 WebDBStart := "WebDB".Start_Roller,
                 WebDBStop := "WebDB".Stop_Roller,
                 WebDBRollerOutput => "WebDB".Output_Roller,
                 RollerDirection => "WebDB".RollerAdjustableOutput.RollerDirection,
                 RollerLinearVelocity => "WebDB".RollerAdjustableOutput.RollerLinearVelocity,
                 RollerRPM => "WebDB".RollerAdjustableOutput.setpointRPM,
                 RollerRPM_Measured => "WebDB".RollerAdjustableOutput.RollerSpeedRPM);
END_REGION

REGION Network 10: Z Axis Missing Layer Detection
   RUNG wire#powerrail
      Contact( "FTON_FirstTurnON".FTON_ZAxisDiagnostic )
      "Z axis missing layer detection_DB"(Mode :=, PrintStarted := "WebDB".PrintingStatus.InPrintStarted, PrintPaused := "WebDB".PrintingStatus.InPrintPaused, PrintEnded := "WebDB".PrintingStatus.InPrintEnded, Z1AxisPosition := "WebDB".Z1Output.ActualPosition, Z1FeedStep := "WebDB".Z1Input.SetValuePosition, Z1Relative := "WebDB".Z1Input.Relative, Z2AxisPosition := "WebDB".Z2Output.ActualPosition, Z2StepSize := "WebDB".Z2Input.SetValuePosition, Z2Relative := "WebDB".Z2Input.Relative, AmountOfLayers :=, MotionMargin :=, CompensationStepSize :=, PrintingStepSize :=, Z1PredictedFinalPositionMinus =>, Z1PredictedFinalPosition =>, Z1PredictedFinalPositionPlus =>, Z2PredictedFinalPositionMinus =>, Z2PredictedFinalPosition =>, Z2PredictedFinalPositionPlus =>, MissingLayerStatus => "WebDB".PrintingStatus.OutMissingLayerDetected, ErrorTime =>)
   END_RUNG
   // the same network as SCL:
   IF "FTON_FirstTurnON".FTON_ZAxisDiagnostic THEN
       "Z axis missing layer detection_DB"(PrintStarted := "WebDB".PrintingStatus.InPrintStarted,   // "Z axis missing layer detection"
                               PrintPaused := "WebDB".PrintingStatus.InPrintPaused,
                               PrintEnded := "WebDB".PrintingStatus.InPrintEnded,
                               Z1AxisPosition := "WebDB".Z1Output.ActualPosition,
                               Z1FeedStep := "WebDB".Z1Input.SetValuePosition,
                               Z1Relative := "WebDB".Z1Input.Relative,
                               Z2AxisPosition := "WebDB".Z2Output.ActualPosition,
                               Z2StepSize := "WebDB".Z2Input.SetValuePosition,
                               Z2Relative := "WebDB".Z2Input.Relative,
                               MissingLayerStatus => "WebDB".PrintingStatus.OutMissingLayerDetected);
   END_IF;
END_REGION
END_ORGANIZATION_BLOCK
